// TwinCAT 3 PLC project PRINCIPAL
// Title: Programa Base 01
// Company: Escarre Automatizacion y Servecios sl
// ProjectVersion: 00_00
// ProgramVersion: 3.1.4023.0
// libraries:
//   EAS PLC, * (ESCARRE AUTOMATIZACION Y SERVICIOS sl)
//   EAS SCADA, * (ESCARRE AUTOMATIZACION Y SERVICIOS sl)
//   Tc2_Standard, * (Beckhoff Automation GmbH)
//   Tc2_SUPS, * (Beckhoff Automation GmbH)
//   Tc2_System, * (Beckhoff Automation GmbH)
//   Tc2_Utilities, * (Beckhoff Automation GmbH)
//   Tc3_Module, * (Beckhoff Automation GmbH)
//   Util, * (System)
// project tree:
//   DUTs/20_HARD/Beckhoff/ Island_Beck.TcDUT (not stored)
//   DUTs/20_HARD/ Hard.TcDUT
//   DUTs/MACHINE/DUT Elements/ dutAIn.TcDUT (not stored), dutAOut.TcDUT (not stored), dutPul.TcDUT, dutPump.TcDUT (not stored), dutValve.TcDUT (not stored)
//   DUTs/MACHINE/DUT System/ _00_GENERAL.TcDUT (not stored), _01_SEG.TcDUT (not stored), _02_TEMP.TcDUT, _03_PRESS.TcDUT (not stored), _04_FILL.TcDUT (not stored), _05_DRAIN.TcDUT, _06_LEVEL.TcDUT, _07_OVERFLOW.TcDUT, _08_CIRC.TcDUT (not stored), _09_CPUMP.TcDUT, _10_TK1.TcDUT, _11_TK2.TcDUT (not stored), _12_INTRO.TcDUT (not stored), _13_T_PREP.TcDUT (not stored), _14_CONSUM.TcDUT, _15_WINCH.TcDUT (not stored), _16_WINCH_X.TcDUT (not stored)
//   DUTs/MACHINE/ Machine.TcDUT
//   DUTs/10_PE/ ATL.TcDUT (not stored)
//   DUTs/10_PE/ELEMENTS/ PE.TcDUT (not stored), PE_COM.TcDUT
//   GVLs/ contants.TcGVL, Gloval_Variables.TcGVL (not stored), Mc.TcGVL (not stored), _Hard.TcGVL, _PE.TcGVL (not stored)
//   / PlcTask.TcTTO
//   POUs/00_Tasks/ ProgramaPrincipal.TcPOU
//   POUs/10_PE/ pComPE.TcPOU (not stored), pPE.TcPOU
//   POUs/20_Hardware/ pHard.TcPOU
//   POUs/30_PLC/30_1 UPS/ UPS.TcPOU
//   POUs/30_PLC/30_2 IO/ pIO.TcPOU
//   POUs/30_PLC/30_3_Config/ConfigSystem/ _00_Config_PE.TcPOU, _14_Config_Consum.TcPOU, _09_Config_CPump.TcPOU (not stored), _05_Config_Drain.TcPOU, _04_Config_Fill.TcPOU (not stored), _06_Config_LEVEL.TcPOU, _07_Config_Overflow.TcPOU (not stored), _03_Config_PRESS.TcPOU, _01_Config_SEG.TcPOU, _02_Config_TEMP.TcPOU (not stored), _10_Config_TK1.TcPOU (not stored), _11_Config_TK2.TcPOU (not stored), _15_Config_Winch.TcPOU, _00_Config_General.TcPOU (not stored)
//   POUs/30_PLC/30_3_Config/ pConfig.TcPOU
//   POUs/30_PLC/30_5_Funcions/Funcions/ F_AVISO.TcPOU, F_CARGA.TcPOU, F_CONTROL_PH.TcPOU, F_DESCARGA.TcPOU, F_DESPRESURIZA.TcPOU, F_DUCHAS.TcPOU (not stored), F_ESPERA.TcPOU (not stored), F_FIN_CICLO.TcPOU, F_FIN_DUCHAS.TcPOU (not stored), F_INTRO_TK2.TcPOU, F_ISOTERMA.TcPOU (not stored), F_LAVADO_CONT.TcPOU (not stored), F_LLENADO.TcPOU (not stored), F_LLENADO_TK2.TcPOU, F_MUESTRA.TcPOU, F_PREP_TK2.TcPOU, F_PRESURIZAR.TcPOU, F_RECIRCULA_TK2.TcPOU (not stored), F_TERMOREG.TcPOU (not stored), F_VACIADO.TcPOU (not stored), F_VACIADO_TK2.TcPOU, F_VELOCIDADES.TcPOU, _00_CIRC_PUMP.TcPOU (not stored), _00_CONSUMS.TcPOU (not stored), _00_GENERALES.TcPOU, _00_GESTION_PUL.TcPOU, _00_PID.TcPOU (not stored), _00_VENT.TcPOU
//   POUs/30_PLC/30_5_Funcions/ pFuctions.TcPOU
//   POUs/30_PLC/30_7 ActvOutputs/Modules/ Z_CIRC.TcPOU, z_CONTROL.TcPOU (not stored), Z_CP.TcPOU (not stored), z_DRAIN.TcPOU, z_FILL.TcPOU (not stored), Z_INTRO.TcPOU (not stored), z_LEVEL.TcPOU, z_OVERFLOW.TcPOU (not stored), z_PRESS.TcPOU, z_TEMP.TcPOU, z_TK1.TcPOU, z_TK2.TcPOU
//   POUs/30_PLC/30_7 ActvOutputs/ pActvOutputs.TcPOU
//   POUs/30_PLC/ ProgramPLC.TcPOU (not stored)
//   POUs/40_Function_Blocks/40_1_Llibreries_FB/ Canvi_Escala.TcPOU (not stored), Polsador.TcPOU, PULS_1S.TcPOU (not stored), TMP_P.TcPOU (not stored)
//   POUs/40_Function_Blocks/FB/Consums/ CONSUMP_00.TcPOU (not stored), KG_vapor_00.TcPOU (not stored), Kwh_00.TcPOU (not stored), Lit_H2O_00.TcPOU (not stored), Tabla_00.TcPOU (not stored)
//   POUs/40_Function_Blocks/FB/FB Duts/ fAI.TcPOU (not stored), fAO.TcPOU (not stored), fCaudal.TcPOU (not stored), fCnt.TcPOU (not stored), fTemp.TcPOU, fValve.TcPOU
//   POUs/40_Function_Blocks/FB/FB%27s_Utils/ fBCntLiters.TcPOU (not stored), fBHorn.TcPOU (not stored), fBPulse1s.TcPOU (not stored), fBUp_Down.TcPOU (not stored), fBWash_TK.TcPOU (not stored), fB_Intro_TK.TcPOU (not stored), fBPumpC.TcPOU (not stored), fBPumpSpeed.TcPOU (not stored), fBTermo.TcPOU (not stored)
//   Project Information/ F_GetCompany.TcPOU, F_GetTitle.TcPOU, F_GetVersion.TcPOU
// real-time tasks:
//   TASK PlcTask: cycle T#10ms, priority 20, ADS port 350
//   TASK PlcTask_1: cycle T#1ms, priority ?, ADS port 351
// I/O:
//   DEVICE Device 1 (EtherCAT), AmsNetId 5.110.215.44.2.1
//     Term 3 (EK1200) [EK1200-5000 EtherCAT Power supply (2A E-Bus)]
//       Term 1 (EL1512) [EL1512 2Ch. +/- Counter 24V, 1kHz]
//       Term 3 (EL1809) [EL1809 16Ch. Dig. Input 24V, 3ms]
//       Term 4 (EL1809) [EL1809 16Ch. Dig. Input 24V, 3ms]
//       Term 5 (EL1809) [EL1809 16Ch. Dig. Input 24V, 3ms]
//       Term 6 (EL2809) [EL2809 16Ch. Dig. Output 24V, 0.5A]
//       Term 7 (EL2809) [EL2809 16Ch. Dig. Output 24V, 0.5A]
//       Term 8 (EL2809) [EL2809 16Ch. Dig. Output 24V, 0.5A]
//       Term 9 (EL3202) [EL3202 2Ch. Ana. Input PT100 (RTD)]
//       Term 10 (EL3054) [EL3054 4Ch. Ana. Input 4-20mA]
//       Term 11 (EL4004) [EL4004 4Ch. Ana. Output 0-10V, 12bit]
//       Term 12 (EL9011) [EL9011 End Terminal]
//   DEVICE Device 4 (NOV-DP-RAM)
// variable links:
//   PRINCIPAL/PRINCIPAL Instance <-> Device 1 (EtherCAT)/Term 3 (EK1200)/Term 1 (EL1512)
//     PlcTask Inputs/pHard.CNT_Device[1] <-> CNT Inputs Channel 1/Counter value
//     PlcTask Inputs/pHard.CNT_Device[2] <-> CNT Inputs Channel 2/Counter value
//   PRINCIPAL/PRINCIPAL Instance <-> Device 1 (EtherCAT)/Term 3 (EK1200)/Term 10 (EL3054)
//     PlcTask Inputs/pHard.AI_Device[{3..6}] <-> AI Standard Channel {1..4}/Value  (4 links)
//   PRINCIPAL/PRINCIPAL Instance <-> Device 1 (EtherCAT)/Term 3 (EK1200)/Term 11 (EL4004)
//     PlcTask Outputs/pHard.AO_Device[{1..4}] <-> AO Outputs Channel {1..4}/Analog output  (4 links)
//   PRINCIPAL/PRINCIPAL Instance <-> Device 1 (EtherCAT)/Term 3 (EK1200)/Term 3 (EL1809)
//     PlcTask Inputs/pHard.DI_Device[{1..16}] <-> Channel {1..16}/Input  (16 links)
//   PRINCIPAL/PRINCIPAL Instance <-> Device 1 (EtherCAT)/Term 3 (EK1200)/Term 4 (EL1809)
//     PlcTask Inputs/pHard.DI_Device[{17..32}] <-> Channel {1..16}/Input  (16 links)
//   PRINCIPAL/PRINCIPAL Instance <-> Device 1 (EtherCAT)/Term 3 (EK1200)/Term 5 (EL1809)
//     PlcTask Inputs/pHard.DI_Device[{33..48}] <-> Channel {1..16}/Input  (16 links)
//   PRINCIPAL/PRINCIPAL Instance <-> Device 1 (EtherCAT)/Term 3 (EK1200)/Term 6 (EL2809)
//     PlcTask Outputs/pHard.DO_Device[{1..16}] <-> Channel {1..16}/Output  (16 links)
//   PRINCIPAL/PRINCIPAL Instance <-> Device 1 (EtherCAT)/Term 3 (EK1200)/Term 7 (EL2809)
//     PlcTask Outputs/pHard.DO_Device[{17..32}] <-> Channel {1..16}/Output  (16 links)
//   PRINCIPAL/PRINCIPAL Instance <-> Device 1 (EtherCAT)/Term 3 (EK1200)/Term 8 (EL2809)
//     PlcTask Outputs/pHard.DO_Device[{33..48}] <-> Channel {1..16}/Output  (16 links)
//   PRINCIPAL/PRINCIPAL Instance <-> Device 1 (EtherCAT)/Term 3 (EK1200)/Term 9 (EL3202)
//     PlcTask Inputs/pHard.AI_Device[1] <-> RTD Inputs Channel 1/Value
//     PlcTask Inputs/pHard.AI_Device[2] <-> RTD Inputs Channel 2/Value

CONFIGURATION PRINCIPAL
    RESOURCE PLC ON TwinCAT3
        TASK PlcTask(INTERVAL := T#10ms, PRIORITY := 20);
        PROGRAM ProgramaPrincipal WITH PlcTask : ProgramaPrincipal;
    END_RESOURCE
END_CONFIGURATION

// ---- DUTs/20_HARD/Hard.TcDUT
TYPE Hard :
STRUCT
	
Beck:ARRAY[1..Max_island_beck] OF Island_beck;

END_STRUCT
END_TYPE

// ---- DUTs/MACHINE/DUT Elements/dutPul.TcDUT
TYPE dutPul :
STRUCT
	xPul:BOOL;		// IN Pulsador
	xPil:BOOL;		// OUT Piloto

END_STRUCT
END_TYPE

// ---- DUTs/MACHINE/DUT System/_02_TEMP.TcDUT
TYPE _02_TEMP :
STRUCT
	///+++++++++++++++++++++++++++++++++++++++
	///HARD
	///+++++++++++++++++++++++++++++++++++++++
	v060_Aper: dutAOut;
	v061_Steam: dutValve;
	v062_Cool: dutValve;
	v063_RetCon: dutValve;
	v064_RecW: dutValve;
	s065_Reg: ftemp;
	s066_Mc: ftemp;
	s067_RetCon: ftemp;
	v068_Purge: dutValve;
	v069_AperCool: dutAout;
	/// Temperatura Maquina 
	rMacTemperature: REAL;
	///Temperatura  Impuesta
	rTempImp: REAL;
	///Señal para abrir retorno de condensados
	xRetCond: BOOL;
	/// PT100 Failure 
	xPT100Failure: BOOL;
	xMaxDifTemp: BOOL;
	///Gradiente por defecto
	iPFDefauldGrad: INT := 0;
	///Tiempo de bomba en m,archa para iniciar termorreg
	iPFTimeOfPumpToRun: INT := 60;
	///Grados para integracion
	iPFGradIntegra: INT := 2;
	///Grados para forzar calentamiento
	iPFGradForzCal: INT := 4;
	///Tiempo de seguridad para conmutacion vapor-frio
	iPFTmpComutac: INT := 30;
	///Grados para conmutacion en Mantenimiento
	iPFGradComutac: INT := 5;
	///PID_ Banda proporcional
	iPFPID_P: INT;
	///PID_ I= Parte integral
	iPFPID_I: INT;
	///PID_ D= Parte Derivada
	iPFPID_D: INT;
	///Temprearatura por debajo no se calienta
	iPFTempMinCool: INT := 45;
	
END_STRUCT
END_TYPE

// ---- DUTs/MACHINE/DUT System/_05_DRAIN.TcDUT
TYPE _05_DRAIN :
STRUCT
	///+++++++++++++++++++++++++++++++++++++++
	///HARD
	///+++++++++++++++++++++++++++++++++++++++
	v015_Grv: dutValve;
	v016_Grv2: dutValve;
	v017_Pump: dutValve;
	s018_LvlHT: dutPul;
	s019_TempHT: dutAIn;
	v020_HT: dutValve;
	v021_WaterHT: dutValve;
	///+++++++++++++++++++++++++++++++++++++++
	///READINGS
	///+++++++++++++++++++++++++++++++++++++++
	iTempHT: INT;
	xLvlHT: BOOL;
	///+++++++++++++++++++++++++++++++++++++++
	///PF - CONFIG
	///+++++++++++++++++++++++++++++++++++++++
	iPFMaxTimeDrain: INT;
	iPFTimeDrenado: INT;
END_STRUCT
END_TYPE

// ---- DUTs/MACHINE/DUT System/_06_LEVEL.TcDUT
TYPE _06_LEVEL :
STRUCT
	///+++++++++++++++++++++++++++++++++++++++
	///HARD
	///+++++++++++++++++++++++++++++++++++++++
	s031_Min: dutPul;
	s032_Perc: dutAIn;
	s033_max: dutPul;
	s034_L3: dutPul;
	s035_L2: dutPul;
	s036_L1: dutPul;
	v038_FillTb: dutValve;
	v039_DrainTb: dutValve;
	///Nivel de la maquina 0..100%
	rLevel: REAL;
	///Nivel 1 de la maquina
	xLvl_1: BOOL;
	///Nivel 2 de la maquina
	xLvl_2: BOOL;
	///Nivel 3 de la maquina
	xLvl_3: BOOL;
	///Nivel minimo de la maquina
	xLvl_min: BOOL;
	///Nivel maximo de la maquina
	xLvl_max: BOOL;
	///Nivel Alto de Recirculación
	xLvl_Wh: BOOL;
	///Nivel Bajoo de Recirculación
	xLvl_Wl: BOOL;
	///Fallo niveles
	xFailLvl: BOOL;
	///+++++++++++++++++++++++++++++++++++++++
	///PF - CONFIG
	///+++++++++++++++++++++++++++++++++++++++
	///Parametros configuracion Nivel analogico de Maquina
	iPFAna_min: INT := 0;
	iPFAna_max: INT := 100;
	///Porcentaje del nivel para bLvl_1
	iPFLvl_1: INT := 20;
	///Porcentaje del nivel para bLvl_2
	iPFLvl_2: INT := 50;
	///Porcentaje del nivel para bLvl_3
	iPFLvl_3: INT := 70;
	///Porcentaje del nivel para bLvl_min
	iPFLvl_min: INT := 0;
	///Porcentaje del nivel para bLvl_max
	iPFLvl_max: INT := 100;
	///Porcentaje del nivel alto de recirculación
	iPFLvl_Wh: INT := 60;
	///Porcentaje del nivel bajo de recirculación
	iPFLvl_Wl: INT := 20;
END_STRUCT
END_TYPE

// ---- DUTs/MACHINE/DUT System/_07_OVERFLOW.TcDUT
TYPE _07_OVERFLOW :
STRUCT
	///+++++++++++++++++++++++++++++++++++++++
	///HARD
	///+++++++++++++++++++++++++++++++++++++++
	v025_Valv: dutValve;
	v026_intrHT: dutValve;
	v027_VentHt: dutValve;
	v028_DrainHT: dutValve;
	v004_WaterInlet: dutValve;
	///Litros de la barcada
	rLit_Batch: REAL;
	///Litros Actuales
	rLit_Actual: REAL;
	///+++++++++++++++++++++++++++++++++++++++
	///CONFIG
	///+++++++++++++++++++++++++++++++++++++++
	iPFTimeFillAuxT: INT := 5;
	iPFTimeCloseAuzT: INT := 5;
	iPFTimeDepAuxT: INT := 5;
	iPFTimeDrainAuxT: INT := 5;
	iPFTimeCloseDrainAuxT: INT := 5;
END_STRUCT
END_TYPE

// ---- DUTs/MACHINE/DUT System/_09_CPUMP.TcDUT
TYPE _09_CPUMP :
STRUCT
	///+++++++++++++++++++++++++++++++++++++++
	///HARD
	///+++++++++++++++++++++++++++++++++++++++
	b450_CircPump: dutPump;
	p451_P_Run: dutPul;
	p452_P_Stop: dutPul;
	p453_P_AutoMan: dutPul;
	p454_P_UpVel: dutPul;
	p455_P_DownVel: dutPul;
	s456_Pote: dutAIn;
	p457_SelRun: dutPul;
	///+++++++++++++++++++++++++++++++++++++++
	///READINGS
	///+++++++++++++++++++++++++++++++++++++++
	rSP_Auto: REAL;
	rSP_Man: REAL;
	rSpeedUF: REAL;
	///+++++++++++++++++++++++++++++++++++++++
	///CONFIG
	///+++++++++++++++++++++++++++++++++++++++
	///++++PF+++
	iPF_AnaMax_UF: INT;
	iPF_AnaMin_UF: INT;
	iPF_AnaMax_perc: INT;
	iPF_AnaMin_perc: INT;
	iPF_SpeedMax_UF: INT;
	iPF_SpeedMin_UF: INT;
END_STRUCT
END_TYPE

// ---- DUTs/MACHINE/DUT System/_10_TK1.TcDUT
TYPE _10_TK1 :
STRUCT
	///+++++++++++++++++++++++++++++++++++++++
	///HARD
	///+++++++++++++++++++++++++++++++++++++++
	v101_Fill: dutValve;
	v102_RetMc: dutValve;
	v103_IntercTK: dutValve;
	b104_Intro: dutPump;
	v105_Drain_Pump: dutValve;
	v106_Drain_grav: dutValve;
	v107_Warm: dutValve;
	p108_Stirrer: dutPump;
	v109_Mixer: dutValve;
	v110_IntecIntro: dutValve;
	v111_Fill_TP: dutValve;
	v112_IntroTK2: dutValve;
	s113_Level: dutAin;
	s114_Temp: dutAin;
	o115_Lev1: dutPul;
	o116_Lev2: dutPul;
	p150_OKprod: dutPul;
	p151_P_Fill: dutPul;
	p152_P_Drain: dutPul;
	P153_P_RetMc: dutPul;
	p154_P_IntroFast: dutPul;
	p155_P_Warm: dutPul;
	p156_P_IntroSlow: dutPul;
	p157_P_Stirrer: dutPul;
	p158_P_Mixer: dutPul;
	p159_P_AutoMan: dutPul;
	p160_P_TK1_TK2: dutPul;
	///+++++++++++++++++++++++++++++++++++++++
	///READINGS
	///+++++++++++++++++++++++++++++++++++++++
	xLvl_min: BOOL;
	xLvl_max: BOOL;
	rLvl: REAL;
	xLvlHighCirc: BOOL;
	xLvlLowCirc: BOOL;
	xLvl_1: BOOL;
	xLvl_2: BOOL;
	xLvl_3: BOOL;
	rQt: REAL;
	rQr: REAL;
	///+++++++++++++++++++++++++++++++++++++++
	///CONFIG
	///+++++++++++++++++++++++++++++++++++++++
	iPFLvlAnaMin: INT;
	iPFLvlAnaMax: INT;
	iPFLvlMin: INT;
	iPFLvlMax: INT;
	iPFDescSonda: INT;
	iPFDreno: INT;
	iPF1rLav: INT;
	iPF2nLav: INT;
	iPF3rLav: INT;
	iPFDifAlarma: INT;
	iPFRetarBomba: INT;
	iPFHighCirc: INT;
	iPFLowCirc: INT;
	/// Volum Tank (Liters)
	iPFVolumTK: INT;
	iPFLvl_1: INT;
	iPFLvl_2: INT;
	iPFLvl_3: INT;
END_STRUCT
END_TYPE

// ---- DUTs/MACHINE/DUT System/_14_CONSUM.TcDUT
TYPE _14_CONSUM :
STRUCT
(*+++++++++++++++++++++++++++++++++++++++*)
(*HARD*)
(*+++++++++++++++++++++++++++++++++++++++*)
	s500_Amperimetre	:dutAin;


	
(*+++++++++++++++++++++++++++++++++++++++*)
(*READINGS*)
(*+++++++++++++++++++++++++++++++++++++++*)

	rLit_Batch		:REAL;		(*Litros de la barcada*)
	rKw_Batch		:REAL; 		(*Kw de la Barcada*)
	rKgStm_Batch	:REAL;		(*Kg de Vapor de la barcada*)
	rAmp			:REAL;		//Corriente de entrada


(*+++++++++++++++++++++++++++++++++++++++*)
(*CONFIG*)
(*+++++++++++++++++++++++++++++++++++++++*)




	
END_STRUCT
END_TYPE

// ---- DUTs/MACHINE/Machine.TcDUT
TYPE Machine :
STRUCT
	///Sistema de Batch
	_00_GENERAL: _00_GENERAL;
	///SEGURIDAD
	_01_SEG: _01_SEG;
	///Sistema de calentamiento
	_02_TEMP: _02_TEMP;
	///Sistema de PRESURITZACIÓ
	_03_PRESS: _03_PRESS;
	///Sistema de llenado
	_04_FILL: _04_FILL;
	///Sistema de Vaciado
	_05_DRAIN: _05_DRAIN;
	///Sistema de Niveles de la maquina
	_06_LEVEL: _06_LEVEL;
	///Sistema de Rebosadero
	_07_OVERFLOW: _07_OVERFLOW;
	///Valvulas de la circulacion
	_08_CIRC: _08_CIRC;
	///Bomba de circulacion
	_09_CPUMP: _09_CPUMP;
	///Tanque 1
	_10_TK1: _10_TK1;
	///Tanque 2
	_11_TK2: _11_TK2;
	///Sistema de Intorduccion
	_12_INTRO: _12_INTRO;
	///Tanque Preparacion
	_13_TPrep: _13_T_PREP;
	///Sistema de Consumos
	_14_CONSUM: _14_CONSUM;
	///Troniquetes
	_15_WINCH: _15_WINCH;
	

	
	
END_STRUCT
END_TYPE

// ---- DUTs/10_PE/ELEMENTS/PE_COM.TcDUT
TYPE PE_COM :
STRUCT
	
(* -------------------------------------------------------------------- *)
(* InfoBarcada *)
	sBatch:STRING[10];			
	diNum_Task:DWORD;
	sCdRecipe:STRING[24];
	sDesc_Recipe:STRING[50];
	sCdCycle:STRING[10];
	sDesc_Cycle:STRING[50];

(* -------------------------------------------------------------------- *)
(* Ordenes PE *)
	xToAutomatic	:BOOL;
	xToManual		:BOOL;
	xToStep			:BOOL;
	xRunCycle		:BOOL;
	xModifiedCycle	:BOOL;
	xStopAlarm		:BOOL;
	xContProg		:BOOL;		 	(*Bit Para continuar programa*)
	xStartTopping	:BOOL;			(*Bit indicacion al iniciar una añadida*)
	xEndTopping		:BOOL;			(*Bit indicacion al finalizar una añadida*)
	xResetStep		:BOOL;			(*Bit indicacion para resetar los tiempos de la funcion al realizar un salto*)
	xReset			:BOOL;
	xResetFunc		:BOOL;
	wNewStep		:WORD;			(*word Per fer un canvi de Pas*)

	
	
(* -------------------------------------------------------------------- *)
(* Dosificacio *)
	
	axDemandDos		: ARRAY [1..max_tanks] OF BOOL;	; 		(* Pedir Dosificacion*)
	aiNumDos		: ARRAY [1..max_tanks] OF WORD;			(* Numero Dosificacion *)
	axOkDemand		: ARRAY [1..max_tanks] OF BOOL;			(* OK Peticion Dosificacion*)	
	axOkDosage		: ARRAY [1..max_tanks] OF BOOL;			(* OK  Dosificacion*)	
	aiTypeDos		: ARRAY [1..max_tanks] OF WORD;	 	  	(* Tipo Dosificacion 1=Man 2=Auto 3=Mixta*)
	axProdMan		: ARRAY [1..max_tanks] OF BOOL;			(* Dosificacion con Producto  Manual **)	
	axErrorDos		: ARRAY [1..max_tanks] OF BOOL;			(* Error Dosificación  **)	
	aiVolumDos		: ARRAY [1..max_tanks] OF DWORD;		(* Volumen dosificat*)
	axTankFree		: ARRAY [1..max_tanks] OF BOOL;			(* Tanque libre *)
	aiPriority		: ARRAY [1..max_tanks] OF WORD;			(* Prioridad*)
	axOnlyDissol	: ARRAY [1..max_tanks] OF BOOL;			(* Solo Disolver*)





	
(* -------------------------------------------------------------------- *)
	
//	No utilizadas:
//	ActivarParalelo:BOOL;
//	DesactivarParalelo:BOOL;



END_STRUCT
END_TYPE

// ---- GVLs/contants.TcGVL
VAR_GLOBAL CONSTANT

(*=======================================	*)
(*			Carregar Constants						*)
(*=======================================	*)
	max_Funcions:WORD:=64;
	max_ParamFunc:WORD:=9;
	max_FinFunc:WORD:=5;
	max_PasCicle:WORD:=256;
	Max_Compatibles:WORD:=32;
	Max_Func_Pas:WORD:=12;
	Max_Alarmes:WORD:=128;
	Max_ParamFixes:WORD:=150;
	Max_DBFiFuncio: WORD:=320 ;				(* Es calcula com    (Max_Funcions*Max_FinFunc)   *)
	Max_ElementsCicle: WORD:=2816 ;		(* Es calcula com    (Max_PasCicle*(Max_ParamFunc+2))  *)
	Max_DBIncompatibles: WORD:=64;			(* Es calcula com    (Max_Compatibles*2)  *)
	Max_Inputs: WORD:=128;
	Max_Outputs: WORD:=128;
	Max_Analog: WORD:=32;
	Num_Prod_Dos:WORD:=10;         					(* Numero maximo de productos en una dosificación*)
	Max_Prod_Dos:WORD:=128;							(* Productos en una dosificadora*)
	Max_Valv_Dos:WORD:=128;							(* Valvulas en una do*)
	Max_Tanks:WORD:=4;
	
	
(*=======================================	*)
(*			Hardware Beckhoff				*)
(*=======================================	*)
	Max_island_beck	:WORD:=5;
	Max_DI_Beck		:WORD:=256;
	Max_DO_Beck		:WORD:=256;
	Max_AI_Beck		:WORD:=32;
	Max_AO_Beck		:WORD:=32;
	Max_CNT_Beck	:WORD:=16;
	
	     
	
END_VAR

// ---- GVLs/_Hard.TcGVL

VAR_GLOBAL 
HARD:Hard;
	

END_VAR

// ---- POUs/00_Tasks/ProgramaPrincipal.TcPOU
PROGRAM ProgramaPrincipal
VAR
	azzz: WORD;
	pols:R_TRIG;
	azzz_ant: WORD;
	cont_scan_2s: WORD;
END_VAR

(*=============================================================*)
(*									++++++++									*)
(*								Programa Principal  							*)
(*									++++++++									*)
(*=============================================================*)

(* Control de run *)
azzz:=azzz+1;
IF azzz>999
	THEN
		azzz:=0;
END_IF


(* -------------------------------------------------------------------------------------------------------------*)
(* 			Pe4																		*)
(* -------------------------------------------------------------------------------------------------------------*)

pComPe();
 


(* -------------------------------------------------------------------------------------------------------------*)
(* 			Gestió del Cicle														*)
(* -------------------------------------------------------------------------------------------------------------*)

pPE();


(* -------------------------------------------------------------------------------------------------------------*)
(* 			Configuracion Hard																		*)
(* -------------------------------------------------------------------------------------------------------------*)


pHard();

(* -------------------------------------------------------------------------------------------------------------*)
(* 			PLC																		*)
(* -------------------------------------------------------------------------------------------------------------*)


ProgramPLC();

END_PROGRAM

// ---- POUs/10_PE/pPE.TcPOU
PROGRAM pPE
VAR PERSISTENT
	Anar1:Salt;
	Anar2:Salt;
	Anar3:Salt;
	Anar4:SaltDePasEnUnCicle;
	Anar5:SaltDePasEnUnCicle;
	Parar:PararTotesLesFuncions;
	PararInici:PararTotesLesFuncions;
	ComprobarSalt:ComprobarFuncionsPas;
	SaltarProximPas:BOOL;
	EsperaSalt:TON;
	AcualitzaDB: CarregarFuncionsActivesAlDB;
	AcualitzaDB2: CarregarFuncionsActivesAlDB;
	PunterCicle0: WORD;
	ferSalt: BOOL;
	FerSaltParalel: BOOL;    (*ordre de salt*)
	EsperaSaltar: TON;
	SaltarPar: BOOL;
	PararTot:PararTotesLesFuncions;
	

(*=========================================================*)	
(*========  GESTIÓ MANUAL  ================================*)	

	Punt_Func: WORD;
	T_Func_Act:T_Funcio;				(* Funcio que indica el punterCicle *)
	FiFuncio:Parar_Func_FiFuncio;
	Incompatibles: Parar_Func_Incomp;
	a: WORD;
	AcualitzaDB3: CarregarFuncionsActivesAlDB;
	

(*=========================================================*)	
	fbFUNBCK: FunBck_v01;
	xFunBck: BOOL;
	tFunBck: Ton;
	tCicloOn: ton;
	rsBatch: Rs;
	
END_VAR
VAR
	run:BOOL;
	inici: Ton;
	fb_UPS_CX8190: FB_S_UPS_CX81xx;
	xCargadas: BOOL;
	xUltimas: BOOL;
	xBackup: BOOL;
	END_VAR

(*==============================================================*)
(*		GESTION REMANENTES PARA CPU CX8190  					*)
(*==============================================================*)
(*
fb_UPS_CX8190(
	sNetID:= , 
	iPLCPort:=851 , 
	tTimeout:= , 
	eUpsMode:= , 
	ePersistentMode:= , 
	tRecoverTime:= , 
	bPowerFailDetect=> , 
	eState=> );

IF _AppInfo.BootDataLoaded THEN
	xCargadas:=TRUE;
	ELSE
		xCargadas:=FALSE;
END_IF

IF _AppInfo.OldBootData THEN
	xUltimas:=FALSE;
	xBackup:=TRUE;
	ELSIF _AppInfo.BootDataLoaded THEN
		xUltimas:=TRUE; 
		xBackup:=FALSE;
END_IF


*)


(*==============================================================*)
(*		GESTION PE												*)
(*==============================================================*)
(*,,,,,,,,,,,,,,,,,,,,,,,,,,,,,,,,,,,,,,,,,,,,,Pasar a manual al reiniciar  ,,,,,,,,,,,,,,,,,,,,,,,,,,,,,,,,,,,,,,,,,,,,,,,	*)
inici(IN:= run, PT:=T#5S , Q=> , ET=> );


IF NOT inici.Q THEN
ATL.PE_COM.xToManual:=TRUE;
ATL.PE.wAutoMan:=1;
ATL.PE_COM.xResetFunc:=TRUE;
PararInici(Estat_F:=est_func );
run:=TRUE;
END_IF



(*,,,,,,,,,,,,,,,,,,,,,,,,,,,,,,,,,,,,,,,,,,,,, Orde de Ejecutar Cicle    ,,,,,,,,,,,,,,,,,,,,,,,,,,,,,,,,,,,,,,,,,,,,,,,,,,,,	*)

IF ATL.PE_COM.xRunCycle
	THEN
		Cicle0:=CicleRebut;
		ATL.PE.wStep :=0;
		ATL.PE.wAutoMan:=2;
		Anar2(
			PasInicial:= 0 ,
			 PasFinal:= ATL.PE.wStep );
		ATL.PE_COM.xRunCycle:= FALSE;
END_IF

(*,,,,,,,,,,,,,,,,,,,,,,,,,,,,,,,,,,,,,,,,,,,,,Orde de Cicle Modificat ,,,,,,,,,,,,,,,,,,,,,,,,,,,,,,,,,,,,,,,,,,,,,,,,	*)
IF ATL.PE_COM.xModifiedCycle
	THEN
		Cicle0:=CicleRebut;
		ATL.PE_COM.xModifiedCycle:=FALSE;
END_IF

(*,,,,,,,,,,,,,,,,,,,,,,,,,,,,,,,,,,,,,,,,,,,,,Orde de Reset ,,,,,,,,,,,,,,,,,,,,,,,,,,,,,,,,,,,,,,,,,,,,,,,,,,,,,,,,,,,,,,,,	*)
IF ATL.PE_COM.xReset
	THEN
		PararTot(Estat_F:=Est_F_PE4 );
		ATL.PE.wStep :=0;
		ATL.PE_COM.xToManual:=TRUE;
		ATL.PE_COM.xReset:=FALSE;
END_IF
(*,,,,,,,,,,,,,,,,,,,,,,,,,,,,,,,,,,,,,,,,,,,,,Orde de Reset ,,,,,,,,,,,,,,,,,,,,,,,,,,,,,,,,,,,,,,,,,,,,,,,,,,,,,,,,,,,,,,,,	*)
IF ATL.PE_COM.xResetFunc
	THEN
		PararTot(Estat_F:=Est_F_PE4 );
		ATL.PE_COM.xResetFunc :=FALSE;
END_IF


(*=============================================================*)
(*=============================================================*)

(*Control si el sistema treballa en MANUAL / AUTOMATIC *)

(*,,,,,,,,,,,,,,,,,,,,,,,,,,,,,,,,,,,,,,,, Canvis d'estat AUTO/MAN ,,,,,,,,,,,,,,,,,,,,,,,,,,,,,,,,,,,,,,,,,,,,,,,,,	*)
(*  Automàtic   *)
IF ((ATL.PE.xPulAuto)(*OR Com_PE.RetardArranc*) OR (ATL.PE_COM.xToAutomatic) OR (ATL.PE.wAutoMan>2))AND(cicle0[1].Pas<>0)
	THEN
		(* Pasar de Manual a Automatic*)
		IF ATL.PE.wAutoMan<=1
			THEN
				Parar(Estat_F:=Est_Func);
				IF ATL.PE.wStep=0
					THEN
						ATL.PE.wStep:=1;
				END_IF
				Anar3(
					PasInicial:= 0 ,
		 			PasFinal:= ATL.PE.wStep );
		END_IF
		ATL.PE.wAutoMan:=2;
		AcualitzaDB
			(EstatFuncions:= Est_Func  ,
			FuncionsActives=>Func_Actives );
END_IF;
		ATL.PE_COM.xToAutomatic:=FALSE;

(*  Manual   *)
IF (ATL.PE.xPulMan) OR (ATL.PE_COM.xToManual) OR (ATL.PE.wAutoMan<1)
	THEN
		(* Pasar d'automatic a manual *)
		IF ATL.PE.wAutoMan>=2
			THEN
				Parar(Estat_F:=Est_Func);
		END_IF
		ATL.PE.wAutoMan:=1;
		ATL.PE_COM.xToManual:=FALSE;
END_IF;


(*=============================================================*)
(* + + + + + + + +  +  + + + + + + + + + + + + + + + + + + + + + + + + + + + + + + + + + *)

(*,,,,,,,,,,,,,,,,,,,,,,,,,,,,,,,,,,,,,,,,,, Gestio Manual,,,,,,,,,,,,,,,,,,,,,,,,,,,,,,,,,,,,,,,,,,,,,,,,,,,,,,,,,,,,,,,,,,,,,	*)

IF ATL.PE.wAutoMan=1
	THEN
(*_____________________________________________________________________________________________________________*)
		Punt_Func:=1;
		REPEAT
			IF (Est_Func[Punt_Func].Actv_Funcio)=(Est_F_PE4[Punt_Func].Actv_Funcio)
			THEN
				(*Igualar valors de les funcions*)
				Est_Func[Punt_Func]:=Est_F_PE4[Punt_Func];
				(*Aumentar el punter*)
				Punt_Func:=Punt_Func+1;
			ELSE
				T_Func_Act:=Config_Func[Punt_Func];
				IF Est_Func[Punt_Func].Actv_Funcio=TRUE
				THEN
					(* Parar la funcio al PLC per fi funcio manual al PE4  *)
					Est_Func[Punt_Func].Actv_Funcio:=FALSE;
				ELSE
					IF (Est_F_PE4[Punt_Func].Actv_Funcio=TRUE)AND(Est_F_PE4_Ant[Punt_Func].Actv_Funcio=TRUE)
					THEN
						(*Parar la funcio al PE4 per que s'ha acabat*)
							Est_F_Pe4[Punt_Func].Actv_Funcio:=FALSE;
					ELSE
						(*=====Activar la funció====*)
						(*Mirar si hi ha alguna funció incompatible amb la nova funció*)
						Incompatibles(
							Funcio:= T_Func_Act.Cd_funcio ,
							DB_Comp:= Func_Comp,
							Estat_F:=Est_Func );
		
						(*Mirar si la funcio nova ha d'acabar alguna funció per Fin Funcion*)
						FiFuncio(
							Tipus_Funcio:= T_Func_Act ,
							Estat_F:= Est_func);
						(*Activar la funció*)
						Est_Func[Punt_Func]:= Est_F_PE4[Punt_Func];
					END_IF
				END_IF
			END_IF
		UNTIL
		Punt_Func>Max_Funcions
		END_REPEAT
		AcualitzaDB3
			(EstatFuncions:= Est_Func  ,
			FuncionsActives=>Func_Actives );
		
		Est_F_PE4_Ant:=Est_F_PE4;
(*_____________________________________________________________________________________________________________*)
		SaltarProximPas:=FALSE;
END_IF


(*=============================================================*)
(* + + + + + + + +  +  + + + + + + + + + + + + + + + + + + + + + + + + + + + + + + + + + *)
(*,,,,,,,,,,,,,,,,,,,,,,,,,,,,,,,,,,,,, Gestio En Autiomatic,,,,,,,,,,,,,,,,,,,,,,,,,,,,,,,,,,,,,,,,,,,,,,,,,,,,,,,,,,,,,	*)


IF ATL.PE.wAutoMan=2
	THEN
		(*__________________Comprobar si cal pasar la seguent PAS_______________________________________________*)
		ComprobarSalt(
			Estat_F:= Est_Func,
			Tipus_F:=Config_Func ,
			FuncionsActives:= Func_Actives,
			AumentaPas=> SaltarProximPas );

		(*__________________Buscar Punter Cicle del pas inicial___________________________________________________*)

	PunterCicle0:=0;
		REPEAT
			PunterCicle0 := PunterCicle0+1;
		UNTIL
			(((Cicle0[PunterCicle0].Pas=ATL.PE.wStep)AND(Cicle0[PunterCicle0+1].Pas<>ATL.PE.wStep)) OR (PunterCicle0>=max_PasCicle))
		END_REPEAT

		(*__________________Fer Canvi de pas _______________________________________________________________*)
		IF SaltarProximPas AND NOT he_C_local
			THEN
				IF NOT(MaquinaEnParalel)
				THEN
				(* ·······················Maquina Single o Paralel desacoplada ··············································································································· *)
				Anar4(
					PasInicial:= ATL.PE.wStep,
		 			PasFinal:= (ATL.PE.wStep + 1) );
				ATL.PE.wStep:=ATL.PE.wStep + 1;
				SaltarProximPas:=FALSE;
				AcualitzaDB(
					EstatFuncions:= Est_Func  ,
					FuncionsActives=>Func_Actives );
				ELSE
				(* ·······················Maquina  En Paralel Acoplada ··························································································································· *)
				(*---------------------------------------------------------------------------------------------------------------------------------------------------------*)
				(*........................Indicar que la maquina local està preparada per pasar de pas..........................:........................................*)
				Preparat_C_local:=TRUE;
				(*........................Ordre de canvi ::::..........::::::::::.........::::::::::.........::::::::::.........::::::::::.........::::::::::.........::::::::::.........::::::::::.........:::::.*)
				(*........................Maquina Master: Actv ordre de canvi de pas.::::::::::.........::::::::::.........::::::::::.........::::::::::.........::::::::::.........:::::.*)
				(* 10/06/2011   preparat per diferents tipus de paralel   *)
				IF tipoparalelo<=2 THEN
					Ordre_C:= Master AND Preparat_C_local AND Preparat_C_S1;
				END_IF
				IF tipoparalelo=3 THEN
					Ordre_C:= Master AND Preparat_C_local AND Preparat_C_S1 AND Preparat_C_S2;
				END_IF
				IF tipoparalelo=4 THEN
					Ordre_C:= Master AND Preparat_C_local AND Preparat_C_S1 AND Preparat_C_S2 AND Preparat_C_S3;
				END_IF
				IF tipoparalelo>=5 THEN
					Ordre_C:= Master AND Preparat_C_local AND Preparat_C_S1 AND Preparat_C_S2 AND Preparat_C_S3 AND Preparat_C_S4;
				END_IF

				(*........................Activar el canvi procedent del master ..........::::::::::.........::::::::::.........::::::::::.........::::::::::.........::::::::::.........:::::.*)
				FerSaltParalel:=Ordre_C_Master AND NOT He_C_local;
				(*"""""""""""""Ordre de saltar,,,,,,,,,,,,,,,,,,,,,,,,,,,,,,,,,,,,,,,,,,,,,,,,,,,,,,,,,,,,,,,,,,,,,,,,,,,,,,,,,,,,,,,,,,,,,,,,,,,,,,,,,,,,,,,,,,,,,,,,,,,,,,,,,,,,,,,,,,,,,,,,,,,,,,,,,,,,,,*)
				IF  SaltarPar THEN
					Anar5(
						PasInicial:= ATL.PE.wStep,
		 				PasFinal:= (ATL.PE.wStep+1) );
					ATL.PE.wStep:=ATL.PE.wStep+1;
					SaltarProximPas:=FALSE;
					AcualitzaDB2(
						EstatFuncions:= Est_Func  ,
						FuncionsActives=>Func_Actives );
				(*........................Marca local  que ja s'ha fet el salt ::::..........::::::::::.........::::::::::.........::::::::::.........::::::::::.........::::::::::.........:::::.*)
					He_C_local:=TRUE;                            (* Marca de salt fet *)
				END_IF
			END_IF
		END_IF
		Est_F_PE4_Ant:=Est_F_PE4;
		Est_F_PE4:=Est_Func;
END_IF

(*Espera per asegurar que no es fa més de un salt de cop*)
EsperaSaltar(IN:= FerSaltParalel, PT:=t#1s , Q=>SaltarPar );

(*........................Maquina Master: Comprobar que tots han fet el canvi:::::::::.........::::::::::.........::::::::::.........::::::::::.........:::::.*)
(* 10/06/2011   preparat per diferents tipus de paralel   *)
IF tipoparalelo<=2 THEN
	Fi_C:= ( Master AND He_C_local AND He_C_S1 )OR( master AND Fi_C AND Preparat_C_S1);
END_IF
IF tipoparalelo=3 THEN
	Fi_C:= ( Master AND He_C_local AND He_C_S1 AND He_C_S2 )OR( master AND Fi_C AND (Preparat_C_S1 OR Preparat_C_S2));
END_IF
IF tipoparalelo=4 THEN
	Fi_C:= ( Master AND He_C_local AND He_C_S1 AND He_C_S2 AND He_C_S3 )OR( master AND Fi_C AND (Preparat_C_S1 OR Preparat_C_S2 OR Preparat_C_S3));
END_IF
IF tipoparalelo>=5 THEN
	Fi_C:= ( Master AND He_C_local AND He_C_S1 AND He_C_S2 AND He_C_S3 AND He_C_S4 )OR( master AND Fi_C AND (Preparat_C_S1 OR Preparat_C_S2 OR Preparat_C_S3 OR Preparat_C_S4));
END_IF



(*........................Fer Reset dels valors per fi de canvi de pas::::::::::::::::::::::::::.........::::::::::.........::::::::::.........::::::::::.........:::::.*)
IF Fi_C_Master OR ATL.PE.wAutoMan<=1 OR NOT(MaquinaEnParalel) THEN
	Preparat_C_local:=FALSE;
	Preparat_C_S1:=FALSE;
	Preparat_C_S2:=FALSE;
	Preparat_C_S3:=FALSE;
	Preparat_C_S4:=FALSE;
	He_C_local:=FALSE;
	He_C_S1:=FALSE;
	He_C_S2:=FALSE;
	He_C_S3:=FALSE;
	He_C_S4:=FALSE;
	Ordre_C:=FALSE;
	Ordre_C_Master:=FALSE;
	FerSaltParalel:=FALSE;
	SaltarPar:=FALSE;
END_IF

(* Reset valors paralel en cas de manual*)
IF ATL.PE.wAutoMan=1
	THEN
	FerSaltParalel:=FALSE;
END_IF

(*,,,,,,,,,,,,,,,,,,,,,,,,,,,,,,,,,,,,,,,,,,,,,Orde de Salt de pas ,,,,,,,,,,,,,,,,,,,,,,,,,,,,,,,,,,,,,,,,,,,,,,,,,,,,,,,,	*)
EsperaSalt(IN:= ATL.PE_COM.xToStep, PT:=T#2S , Q=>ferSalt , ET=> );
IF ferSalt 
	THEN
		Parar(Estat_F:= Est_Func );
		Anar1(
			PasInicial:= 0 ,
			PasFinal:= ATL.PE_COM.wNewStep );
		ATL.PE.wStep:=ATL.PE_COM.wNewStep;
		ATL.PE_COM.xResetStep:=TRUE;
		ATL.PE_COM.xToStep:= FALSE;
END_IF
AcualitzaDB(
	EstatFuncions:= Est_Func  ,
	FuncionsActives=>Func_Actives );


(*=====================================================================================================================================*)
(* INDICACIONS AUTO MAN*)

ATL.PE.xMan := ATL.PE.wAutoMan= 1  ;
ATL.PE.xAuto := ATL.PE.wAutoMan= 2  ;

(*=====================================================================================================================================*)
(*CALCULO DURACION PASO*)
fbFUNBCK(funcioBck=>xFunBck );
tFunBck(IN:=xFunBck , PT:=T#10D );
ATL.PE.wTStep := REAL_TO_WORD((TIME_TO_REAL(tFunBck.ET))/1000.0); (*expresado en segundos*)
(*=====================================================================================================================================*)
(*CALCULO DURACION BARCADA*)
rsBatch(SET:=ATL.PE.xStartBatch , RESET1:=ATL.PE.xEndBatch );
tCicloOn(IN:= rsBatch.Q1, PT:=T#10D );
ATL.PE.wTBatch:= REAL_TO_WORD((TIME_TO_REAL(tCicloOn.ET))/60000.0);(*expresado en minutos*)
(*=====================================================================================================================================*)

END_PROGRAM

// ---- POUs/20_Hardware/pHard.TcPOU
PROGRAM pHard
VAR
	DI_Device AT %I*: ARRAY[1..Max_DI_Beck] OF BOOL;
	DO_Device AT %Q*: ARRAY[1..Max_DO_Beck] OF BOOL;
	AI_Device AT %I*: ARRAY[1..Max_AI_Beck] OF INT;
	AO_Device AT %Q*: ARRAY[1..Max_AO_Beck] OF INT;
	CNT_Device AT %I*: ARRAY[1..Max_CNT_Beck] OF UDINT;
	Borrar:BOOL;
	
	iPunt: WORD;
END_VAR


(*==============================================================
1001= DI
1002= DO
1003= AI 0..10V
1004= AI 4..20mA
1005= AO 0..10V
1006= AO 4..20mA
1007= AI pt-100
1008= CNT

===================================================================*)

(*==============================================================
1001= DI
1002= DO
1003= AI 0..10V
1004= AI 4..20mA
1005= AO 0..10V
1006= AO 4..20mA
1007= AI pt-100
1008= CNT

===================================================================*)(*-------------------------------------------------------------------------*)
(*CArgar configuracion Beckhoff a la variable HArd*)
(*-------------------------------------------------------------------------*)
(*DI*)
iPunt:=1;
WHILE ipunt< Max_DI_Beck+1
	DO
	hard.Beck[1].DIN[iPunt]:=DI_Device[ipunt];
	iPunt:=iPunt+1;
END_WHILE
(*-------------------------------------------------------------------------*)
(*DO*)
iPunt:=1;
WHILE ipunt< Max_DO_Beck+1
	DO
	DO_Device[ipunt]:=hard.Beck[1].DOUT[iPunt];
	iPunt:=iPunt+1;
END_WHILE
(*-------------------------------------------------------------------------*)
(*AI*)
iPunt:=1;
WHILE ipunt< Max_AI_Beck+1
	DO
	hard.Beck[1].AIN[iPunt]:=AI_Device[ipunt];
	iPunt:=iPunt+1;
END_WHILE
(*-------------------------------------------------------------------------*)
(*AO*)
Borrar:=TRUE;
iPunt:=1;
WHILE ipunt< Max_AO_Beck+1
	DO
	AO_Device[ipunt]:=REAL_TO_INT(hard.Beck[1].AOUT[iPunt]);
	iPunt:=iPunt+1;
END_WHILE

(*-------------------------------------------------------------------------*)
(*CNT*)
iPunt:=1;
WHILE ipunt< Max_CNT_Beck+1
	DO
	hard.Beck[1].CNT[iPunt]:=CNT_Device[ipunt];
	iPunt:=iPunt+1;
END_WHILE
(*-------------------------------------------------------------------------*)

END_PROGRAM

// ---- POUs/30_PLC/30_1 UPS/UPS.TcPOU
PROGRAM UPS
VAR
	run:BOOL;
	
	fb_UPS_CX8190: FB_S_UPS_CX81xx;
	fb_UPS_CX9020: FB_S_UPS_CX9020_U900;
	xCargadas: BOOL;
	xUltimas: BOOL;
	xBackup: BOOL;
END_VAR

(*==============================================================*)
(*		GESTION REMANENTES PARA CPU CX8190 O CX9020 					*)
(*==============================================================*)
(*
fb_UPS_CX8190(
	sNetID:= , 
	iPLCPort:=851 , 
	tTimeout:= , 
	eUpsMode:= , 
	ePersistentMode:= , 
	tRecoverTime:= , 
	bPowerFailDetect=> , 
	eState=> );*)
	
	fb_UPS_CX9020(
	sNetID:= , 
	iPLCPort:=851 , 
	tTimeout:= , 
	eUpsMode:= , 
	ePersistentMode:= , 
	tRecoverTime:= , 
	bPowerFailDetect=> , 
	eState=> );

IF _AppInfo.BootDataLoaded THEN
	xCargadas:=TRUE;
	ELSE
		xCargadas:=FALSE;
END_IF

IF _AppInfo.OldBootData THEN
	xUltimas:=FALSE;
	xBackup:=TRUE;
	ELSIF _AppInfo.BootDataLoaded THEN
		xUltimas:=TRUE; 
		xBackup:=FALSE;
END_IF

END_PROGRAM

// ---- POUs/30_PLC/30_2 IO/pIO.TcPOU
PROGRAM pIO
VAR
	Cargar: INT;
	aaa: INT;
	MANUAL: INT;
	AA: REAL;
END_VAR


(*======================================================================*)
(*			COUNTER INPUTS												*)
(*======================================================================*)
MC._04_FILL.s010_Flowm.iCnt  			:= hard.Beck[1].CNT[1];
//MC.CONSUM.s500_Amperimetre.R	:= hard.Beck[1].CNT[2];
(*======================================================================*)
(*			DIGITAL INPUTS												*)
(*======================================================================*)
(*========= MODULO 2 ===================================================*)

Mc._00_GENERAL.p400_PMAn.xPul			:= hard.Beck[1].DIN[1];
Mc._00_GENERAL.p401_PAuto.xPul			:= hard.Beck[1].DIN[2];
Mc._00_GENERAL.p402_StopAlarm.xPul		:= hard.Beck[1].DIN[3];
Mc._00_GENERAL.p403_ContProg.xPul		:= hard.Beck[1].DIN[4];
Mc._00_GENERAL.p411_FailPump.xPul		:= hard.Beck[1].DIN[5];  				 
Mc._01_SEG.s420_MaxPresTemp.xPul		:= hard.Beck[1].DIN[6];
Mc._01_SEG.s421_BloqValv.xPul			:= hard.Beck[1].DIN[7];
Mc._06_LEVEL.s031_Min.xPul				:= hard.Beck[1].DIN[8];
Mc._01_SEG.s422_McClose.xPul			:= hard.Beck[1].DIN[9];
//Mc._00_GENERAL.p400_PMAn.xPul	 		:= hard.Beck[1].DIN[10];
mc._06_LEVEL.s036_L1.xPul				:= hard.Beck[1].DIN[11];
Mc._06_LEVEL.s035_L2.xPul				:= hard.Beck[1].DIN[12];
Mc._06_LEVEL.s034_L3.xPul				:= hard.Beck[1].DIN[13];
Mc._15_WINCH.W[1].s07_Tangle.xPul		:= hard.Beck[1].DIN[14];
Mc._15_WINCH.W[2].s07_Tangle.xPul		:= hard.Beck[1].DIN[15];					
//Mc._15_WINCH.W[1].p00_Winch.xInCons	:= hard.Beck[1].DIN[16];			  

(*========= MODULO 3 ===================================================*)

Mc._09_CPUMP.p451_P_Run.xPul		:= hard.Beck[1].DIN[17];	
Mc._09_CPUMP.p452_P_Stop.xPul			:= hard.Beck[1].DIN[18];
Mc._09_CPUMP.b450_CircPump.xInCons		:=true;//:= hard.Beck[1].DIN[19];
Mc._09_CPUMP.p453_P_AutoMan.xPul		:= hard.Beck[1].DIN[20];
Mc._09_CPUMP.p455_P_DownVel.xPul		:= hard.Beck[1].DIN[21]; 
Mc._09_CPUMP.p454_P_UpVel.xPul			:= hard.Beck[1].DIN[22];	
Mc._15_WINCH.W[1].p01_Run.xPul			:= hard.Beck[1].DIN[23];
Mc._15_WINCH.W[1].p02_Rev.xPul			:= hard.Beck[1].DIN[24];
Mc._15_WINCH.W[1].P03_AutoMan.xPul		:= hard.Beck[1].DIN[25];
Mc._15_WINCH.W[1].p06_DwnVel.xPul		:= hard.Beck[1].DIN[26];
Mc._15_WINCH.W[1].p05_UpVel.xPul		:= hard.Beck[1].DIN[27];
Mc._15_WINCH.W[1].s11_FindSeam.xPul		:= hard.Beck[1].DIN[28];
Mc._15_WINCH.W[1].s10_ControlSeam.xPul	:= hard.Beck[1].DIN[29];
Mc._15_WINCH.W[2].s10_ControlSeam.xPul	:= hard.Beck[1].DIN[30]; 
Mc._15_WINCH.W[2].s11_FindSeam.xPul		:= hard.Beck[1].DIN[31];
Mc._15_WINCH.W[2].p01_Run.xPul			:= hard.Beck[1].DIN[32]; 

(*========= MODULO 4 ===================================================*)

Mc._12_INTRO.b056_Intro_Pump.xInCons	:= hard.Beck[1].DIN[33];	
Mc._10_TK1.p150_OKprod.xPul				:= hard.Beck[1].DIN[34];
Mc._10_TK1.p151_P_Fill.xPul				:= hard.Beck[1].DIN[35];
Mc._10_TK1.P153_P_RetMc.xPul			:= hard.Beck[1].DIN[36];
Mc._10_TK1.p152_P_Drain.xPul			:= hard.Beck[1].DIN[37]; 
Mc._10_TK1.p154_P_IntroFast.xPul		:= hard.Beck[1].DIN[38];	
Mc._03_PRESS.s072_Chargr.xPul			:= hard.Beck[1].DIN[39];
Mc._03_PRESS.s073_Discharge.xPul		:= hard.Beck[1].DIN[40];
//		:= hard.Beck[1].DIN[41];
//		:= hard.Beck[1].DIN[42];
//		:= hard.Beck[1].DIN[43];
//		:= hard.Beck[1].DIN[44];
//		:= hard.Beck[1].DIN[45];
//		:= hard.Beck[1].DIN[46]; 
//		:= hard.Beck[1].DIN[47];
Mc._11_TK2.p250_OKprod.xPul				:= hard.Beck[1].DIN[48];
(*======================================================================*)
(*			DIGITAL OUTPUTS												*)
(*======================================================================*)
(*========= MODULO 5 ===================================================*)

hard.Beck[1].DOUT[1] := 			MC._00_GENERAL.p400_PMAn.xPil;
hard.Beck[1].DOUT[2] := 			MC._00_GENERAL.p401_PAuto.xPil;
hard.Beck[1].DOUT[3] := 			MC._00_GENERAL.p404_Alarm.xPil;
hard.Beck[1].DOUT[4] := 			MC._00_GENERAL.p405_Horn.xPil;
hard.Beck[1].DOUT[5] := 			MC._03_PRESS.v070_Vent.xOpen;
hard.Beck[1].DOUT[6] := 			MC._04_FILL.v002_Hot.xOpen;
hard.Beck[1].DOUT[7] := 			MC._04_FILL.v001_Cool.xOpen;
hard.Beck[1].DOUT[8] := 			MC._04_FILL.v003_Hard.xOpen;
hard.Beck[1].DOUT[9] := 			MC._05_DRAIN.v015_Grv.xOpen;
hard.Beck[1].DOUT[10] := 			MC._07_OVERFLOW.v025_Valv.xOpen;
hard.Beck[1].DOUT[11] := 			MC._02_TEMP.v061_Steam.xOpen;
hard.Beck[1].DOUT[12] := 			MC._02_TEMP.v062_Cool.xOpen;
hard.Beck[1].DOUT[13] := 			MC._02_TEMP.v063_RetCon.xOpen;
hard.Beck[1].DOUT[14] := 			MC._02_TEMP.v064_RecW.xOpen;
//hard.Beck[1].DOUT[15] := 			;
hard.Beck[1].DOUT[16] := 			MC._04_FILL.v006_InterMc.xOpen;

(*========= MODULO 6 ===================================================*)

hard.Beck[1].DOUT[17] := 			MC._09_CPUMP.b450_CircPump.xRUN;
hard.Beck[1].DOUT[18] := 			MC._15_WINCH.W[1].p00_Winch.xRUN;
//hard.Beck[1].DOUT[19] := 			MC._15_WINCH.W[1].p00_Winch.;
hard.Beck[1].DOUT[20] := 			MC._15_WINCH.W[1].p08_PilTangle.xPil;
hard.Beck[1].DOUT[21] := 			MC._15_WINCH.W[2].p00_Winch.xRUN;
//hard.Beck[1].DOUT[22] := 			MC._10_TK1.v103_IntercTK.xOpen;
hard.Beck[1].DOUT[23] := 			MC._15_WINCH.W[2].p08_PilTangle.xPil;
hard.Beck[1].DOUT[24] := 			MC._12_INTRO.b056_Intro_Pump.xRUN;
hard.Beck[1].DOUT[25] := 			MC._10_TK1.p150_OKprod.xPil;
hard.Beck[1].DOUT[26] := 			MC._10_TK1.v101_Fill.xOpen;
hard.Beck[1].DOUT[27] := 			MC._10_TK1.v102_RetMc.xOpen;
hard.Beck[1].DOUT[28] := 			MC._10_TK1.v106_Drain_grav.xOpen;
hard.Beck[1].DOUT[29] := 			MC._12_INTRO.v050_Fast.xOpen;
hard.Beck[1].DOUT[30] := 			MC._12_INTRO.v051_Slow.xOpen;
hard.Beck[1].DOUT[31] := 			MC._10_TK1.v109_Mixer.xOpen;
hard.Beck[1].DOUT[32] := 			MC._10_TK1.v107_Warm.xOpen;

(*========= MODULO 7 ===================================================*)

hard.Beck[1].DOUT[33] := 			MC._03_PRESS.v071_Load.xOpen;
hard.Beck[1].DOUT[34] := 			MC._03_PRESS.v074_Unload.xOpen;
hard.Beck[1].DOUT[35] := 			MC._07_OVERFLOW.v004_WaterInlet.xOpen;
hard.Beck[1].DOUT[36] := 			MC._08_CIRC.v044_Spray.xOpen;
hard.Beck[1].DOUT[37] := 			MC._05_DRAIN.v017_Pump.xOpen;
hard.Beck[1].DOUT[38] := 			MC._02_TEMP.v068_Purge.xOpen;
hard.Beck[1].DOUT[39] := 			MC._08_CIRC.v041_InPump.xOpen;
hard.Beck[1].DOUT[40] := 			MC._10_TK1.v103_IntercTK.xOpen;
hard.Beck[1].DOUT[41] := 			MC._11_TK2.p250_OKprod.xPil;
hard.Beck[1].DOUT[42] := 			MC._11_TK2.v201_Fill.xOpen;
hard.Beck[1].DOUT[43] := 			MC._11_TK2.v202_RetMc.xOpen;
hard.Beck[1].DOUT[44] := 			MC._11_TK2.v206_Drain_grav.xOpen;	
hard.Beck[1].DOUT[45] := 			MC._11_TK2.v203_IntercTK.xOpen;
hard.Beck[1].DOUT[46] := 			MC._11_TK2.v209_Mixer.xOpen;
hard.Beck[1].DOUT[47] := 			MC._11_TK2.v207_Warm.xOpen;;	
hard.Beck[1].DOUT[48] := 			MC._11_TK2.b204_Intro.XRun;

(*========= MODULO 8 ===================================================*)
MC._02_TEMP.s065_Reg.iAnalog		:=  hard.Beck[1].AIN[1];
//									:=  hard.Beck[1].AIN[2];		
	
(*========= MODULO 9 ===================================================*)
MC._06_LEVEL.s032_Perc.iAnalog		:=	hard.Beck[1].AIN[3];				
MC._10_TK1.s113_Level.iAnalog		:=  hard.Beck[1].AIN[4]; 	
MC._11_TK2.s213_Level.iAnalog		:=MANUAL;//:=	hard.Beck[1].AIN[5];	
Mc._03_PRESS.s075_Sensor.iAnalog	:=	hard.Beck[1].AIN[6];

(*========= MODULO 13 ==================================================*)
hard.Beck[1].AOUT[1]:=				REAL_TO_INT (Z_TEMP.rOutRegTemp);
hard.Beck[1].AOUT[2]:=				REAL_TO_INT (Z_CP.rOutAnalogVelPump);
//hard.Beck[1].AOUT[3]:=				REAL_TO_INT (_15_WINCH.W[1].rSpeedUF);
//hard.Beck[1].AOUT[4]:=				REAL_TO_INT (_15_WINCH.W[2].rSpeedUF);

END_PROGRAM

// ---- POUs/30_PLC/30_7 ActvOutputs/Modules/z_TEMP.TcPOU
PROGRAM z_TEMP

VAR
	rOutRegTemp: REAL;
END_VAR

(*-------------------------------------------------------------------------------------------------------*)
(*v061  Valvula de vapor*)
mc._02_TEMP.v061_Steam.xOpen:= F_TERMOREG.Z_xVapor OR
								F_ISOTERMA.Z_xVapor;

(*-------------------------------------------------------------------------------------------------------*)
(*v062  Valvula de enfriamiento*)
mc._02_TEMP.v062_Cool.xOpen:= F_TERMOREG.z_xEnfria OR
								F_ISOTERMA.z_xEnfria;

(*-------------------------------------------------------------------------------------------------------*)
(*v060  Apertura ValvulaModulante*)
//calentar temo
IF Mc._02_TEMP.v061_Steam.xOpen AND F_TERMOREG.xActv THEN
	Mc._02_TEMP.v060_Aper.rValue:= F_TERMOREG.z_rApertVapor;
END_IF

//calentar ISOTERMA
IF Mc._02_TEMP.v061_Steam.xOpen AND F_ISOTERMA.xActv THEN
	mc._02_TEMP.v060_Aper.rValue:= F_ISOTERMA.z_rApertVapor;
END_IF

//ENFRIAR TERMO
IF Mc._02_TEMP.v062_Cool.xOpen AND F_TERMOREG.xActv THEN
	MC._02_TEMP.v060_Aper.rValue:= F_TERMOREG.z_rApertEnfria;
END_IF

//ENFRIAR ISOTERMA
IF
	MC._02_TEMP.v062_Cool.xOpen AND F_ISOTERMA.xActv THEN
	MC._02_TEMP.v060_Aper.rValue:= F_ISOTERMA.z_rApertEnfria;
END_IF

//OUTPUT Regulacion Temperatura

rOutRegTemp:= Canvi_Escala(
				In:= mc._02_TEMP.v060_Aper.rValue, 
				In_Min:= 0, 
				In_Max:= 1, 
				Out_Min:= 0, 
				Out_Max:= 32675);
	

(*-------------------------------------------------------------------------------------------------------*)
(*v063 Retorno condensados*)
mc._02_TEMP.v063_RetCon.xOpen:= F_TERMOREG.z_xRetonoCond;

(*-------------------------------------------------------------------------------------------------------*)

END_PROGRAM

// ---- POUs/30_PLC/30_3_Config/ConfigSystem/_00_Config_PE.TcPOU
PROGRAM _00_Config_PE
VAR
	A: INT;
END_VAR

A:=A+1;

(*-------------------------------------------------------------------------------------------------------*)
(*_00_General*)
Mc._00_GENERAL.iPFTempAlta		:= WORD_TO_INT(PF[2]);		(*Temperatura para marcar temperatua alta*)

(*-------------------------------------------------------------------------------------------------------*)
(*_01_seg*)
Mc._01_SEG.iPFPresMin := 0 ;    (*FALTA DEFINIR*)
Mc._01_SEG.iPFMcMaxiTemper		:= WORD_TO_INT(PF[1]);		(*PF Maxima Temperatura Maquina*)
Mc._01_SEG.iPFTempCloseVent 	:= WORD_TO_INT(PF[3]);		(*PF Temperatura Cierra Respiradero*)
Mc._01_SEG.iPFTempBloqValv  	:= WORD_TO_INT(PF[2]);		(*PF Temperatura Bloqueo Valvulas*)
		
(*-------------------------------------------------------------------------------------------------------*)
(*_02_TEMP*)
Mc._02_TEMP.iPFDefauldGrad		:= WORD_TO_INT(PF[81]);
Mc._02_TEMP.iPFTimeOfPumpToRun	:= WORD_TO_INT(PF[82]);
Mc._02_TEMP.iPFGradIntegra		:= WORD_TO_INT(PF[83]);
Mc._02_TEMP.iPFGradForzCal		:= WORD_TO_INT(PF[84]);
Mc._02_TEMP.iPFTmpComutac		:= WORD_TO_INT(PF[85]);
Mc._02_TEMP.iPFGradComutac		:= WORD_TO_INT(PF[86]);
Mc._02_TEMP.iPFPID_P			:= WORD_TO_INT(PF[87]);
Mc._02_TEMP.iPFPID_I			:= WORD_TO_INT(PF[88]);
Mc._02_TEMP.iPFPID_D			:= WORD_TO_INT(PF[89]);
Mc._02_TEMP.iPFTempMinCool		:= WORD_TO_INT(PF[90]);


(*-------------------------------------------------------------------------------------------------------*)
(*_03_PRESS*)
Mc._03_PRESS.IPF_FS_Press 		:= WORD_TO_INT(PF[36]);
Mc._03_PRESS.iPFPresLoad 		:= WORD_TO_INT(PF[37]);
Mc._03_PRESS.IPFPresUnload 	 	:= WORD_TO_INT(PF[38]);
Mc._03_PRESS.IPFPresSeg  		:= WORD_TO_INT(PF[39]);
Mc._03_PRESS.IPFTimeOKPresSeg	:= WORD_TO_INT(PF[40]);
Mc._03_PRESS.IPFTimeDelayVent	:= WORD_TO_INT(PF[41]);

(*-------------------------------------------------------------------------------------------------------*)
(*_04_FILL*)
Mc._04_FILL.iPFFrec			  	:= WORD_TO_INT(PF[19]);		(*PF Frecuencia maxima caudalimetro*)
Mc._04_FILL.iPFFlowMax		  	:= WORD_TO_INT(PF[20]);		(*PF Caudal a la freq maxima*)
Mc._04_FILL.iPFTmClcFlow	  	:= WORD_TO_TIME(1000*PF[21]); (*PF Tiempo para el calculo de lcaudal*)
Mc._04_FILL.IPFMaxFillTime		:= PF[23];

(*-------------------------------------------------------------------------------------------------------*)
(*_05_DRAIN*)
Mc._05_DRAIN.iPFMaxTimeDrain	:= WORD_TO_INT(PF[27]) ;    //Maximo tiempo para Vaciado en seg.
Mc._05_DRAIN.iPFTimeDrenado		:= WORD_TO_INT(PF[28]) ;    //Tiempo de drenado maq. en seg.

(*-------------------------------------------------------------------------------------------------------*)
(*_06_LEVEL*)
Mc._06_LEVEL.iPFAna_min			:= WORD_TO_INT(PF[10]);		(*Ajuste minimo nivel analogico*)	
Mc._06_LEVEL.iPFAna_max			:= WORD_TO_INT(PF[11]);		(*Ajuste maximo nivel analogico*)	

Mc._06_LEVEL.iPFLvl_1			:= WORD_TO_INT(PF[14]);		(*Porcentaje del nivel para bLvl_1*)
Mc._06_LEVEL.iPFLvl_2			:= WORD_TO_INT(PF[15]);		(*Porcentaje del nivel para bLvl_2*)
Mc._06_LEVEL.iPFLvl_3			:= WORD_TO_INT(PF[16]);		(*Porcentaje del nivel para bLvl_3*)
Mc._06_LEVEL.iPFLvl_min			:= WORD_TO_INT(PF[17]);		(*Porcentaje del nivel para bLvl_min*)
Mc._06_LEVEL.iPFLvl_max			:= WORD_TO_INT(PF[18]);		(*Porcentaje del nivel para bLvl_max*)

Mc._06_LEVEL.iPFLvl_Wh			:= WORD_TO_INT(PF[12]);		(*Porcentaje del nivel bajo del lavado continuo*)
Mc._06_LEVEL.iPFLvl_Wl			:= WORD_TO_INT(PF[13]);		(*Porcentaje del nivel alto del lavado continuo*)

(*-------------------------------------------------------------------------------------------------------*)
(*_07_OVERFLOW*)
MC._07_OVERFLOW.iPFTimeFillAuxT			:= WORD_TO_INT(PF[30]);		(*Tiempo llena tank auxiliar*)	
MC._07_OVERFLOW.iPFTimeCloseAuzT		:= WORD_TO_INT(PF[31]);		(*Tiempo Fin Llenado tank auxiliar*)	
MC._07_OVERFLOW.iPFTimeDepAuxT			:= WORD_TO_INT(PF[32]);		(*Tiempo despressuriza tank aux*)	 
MC._07_OVERFLOW.iPFTimeDrainAuxT		:= WORD_TO_INT(PF[33]);		(*Tiempo Vaciado tank aux*)	
MC._07_OVERFLOW.iPFTimeCloseDrainAuxT	:= WORD_TO_INT(PF[34]);		(*Tiempo fin vaciado tank aux*)	

(*-------------------------------------------------------------------------------------------------------*)
(*_10_TK1*)
Mc._10_TK1.iPFLvlAnaMin 		:= WORD_TO_INT(PF[50]) ;
Mc._10_TK1.iPFLvlAnaMax 		:= WORD_TO_INT(PF[51]) ;
Mc._10_TK1.iPFLvlMin			:= WORD_TO_INT(PF[52]) ;
Mc._10_TK1.iPFLvlMax			:= WORD_TO_INT(PF[53]) ;
Mc._10_TK1.iPFDescSonda			:= WORD_TO_INT(PF[54]) ;
Mc._10_TK1.iPFDreno				:= WORD_TO_INT(PF[55]) ;
Mc._10_TK1.iPF1rLav				:= WORD_TO_INT(PF[56]) ;
Mc._10_TK1.iPF2nLav				:= WORD_TO_INT(PF[57]) ;
Mc._10_TK1.iPF3rLav				:= WORD_TO_INT(PF[58]) ;
Mc._10_TK1.iPFDifAlarma			:= WORD_TO_INT(PF[59]) ;
Mc._10_TK1.iPFRetarBomba		:= WORD_TO_INT(PF[60]) ;
Mc._10_TK1.iPFLowCirc			:= WORD_TO_INT(PF[61]) ;
Mc._10_TK1.iPFHighCirc			:= WORD_TO_INT(PF[62]) ;
Mc._10_TK1.iPFLvl_1				:= WORD_TO_INT(PF[63]) ;
Mc._10_TK1.iPFLvl_2				:= WORD_TO_INT(PF[64]) ;
Mc._10_TK1.iPFLvl_3				:= WORD_TO_INT(PF[65]) ;

(*-------------------------------------------------------------------------------------------------------*)
(*_11_TK2*)
Mc._11_TK2.iPFLvlAnaMin 		:= WORD_TO_INT(PF[70]) ;
Mc._11_TK2.iPFLvlAnaMax 		:= WORD_TO_INT(PF[71]) ;
Mc._11_TK2.iPFLvlMin			:= WORD_TO_INT(PF[72]) ;
Mc._11_TK2.iPFLvlMax			:= WORD_TO_INT(PF[73]) ;
Mc._11_TK2.iPFDescSonda			:= WORD_TO_INT(PF[74]) ;
Mc._11_TK2.iPFDreno				:= WORD_TO_INT(PF[75]) ;
Mc._11_TK2.iPF1rLav				:= WORD_TO_INT(PF[76]) ;
Mc._11_TK2.iPF2nLav				:= WORD_TO_INT(PF[77]) ;
Mc._11_TK2.iPF3rLav				:= WORD_TO_INT(PF[78]) ;
Mc._11_TK2.iPFDifAlarma			:= WORD_TO_INT(PF[79]) ;
Mc._11_TK2.iPFRetarBomba		:= WORD_TO_INT(PF[80]) ;
Mc._11_TK2.iPFLowCirc			:= WORD_TO_INT(PF[95]) ;
Mc._11_TK2.iPFHighCirc			:= WORD_TO_INT(PF[96]) ;
Mc._11_TK2.iPFLvl_1				:= WORD_TO_INT(PF[97]) ;
Mc._11_TK2.iPFLvl_2				:= WORD_TO_INT(PF[98]) ;
Mc._11_TK2.iPFLvl_3				:= WORD_TO_INT(PF[99]) ;

(*-------------------------------------------------------------------------------------------------------*)
(*_15_WINCH*)
Mc._15_WINCH.iPFWinchToStop		:= WORD_TO_INT(PF[31]); //Torniquete a parar en muestra (0= el primero que pase/ X= toniquete X)


Mc._15_WINCH.iPFNumSeam			:= WORD_TO_INT(PF[32]);//Numero de cuerdas
	IF Mc._15_WINCH.iPFNumSeam=0 
	THEN
	Mc._15_WINCH.iPFNumSeam:=1;
END_IF

Mc._15_WINCH.iPFNumWinch		:= WORD_TO_INT(PF[33]);//Numero de torniquetes
	IF Mc._15_WINCH.iPFNumWinch=0 
	THEN
	Mc._15_WINCH.iPFNumWinch:=1;
END_IF

Mc._15_WINCH.iPFDelayRunWinch	:= WORD_TO_INT(PF[34]);//Retraso arranque Torniquete
Mc._15_WINCH.iPFPercentWinch	:= WORD_TO_INT(PF[35]);//Porcentaje para Alarna de cuerda Parada
Mc._15_WINCH.iPFWinchMaxSpeed	:= WORD_TO_INT(PF[30]);//Velocidad Maxima torniquete
Mc._15_WINCH.iPFFactPulTor		:= WORD_TO_INT(Pf[29]);//Factor pulsadores
Mc._15_WINCH.iPFTimeMaxRope		:= WORD_TO_INT(Pf[42]);//Tiempo Maximo paso cuerda

END_PROGRAM

// ---- POUs/30_PLC/30_3_Config/ConfigSystem/_14_Config_Consum.TcPOU
PROGRAM _14_Config_Consum


(*s 500 sensor ampers para consumo*)
Mc._14_CONSUM.s500_Amperimetre.rAna_min:=0;
Mc._14_CONSUM.s500_Amperimetre.rAna_max:=37000;
Mc._14_CONSUM.s500_Amperimetre.rUf_min:=0;
Mc._14_CONSUM.s500_Amperimetre.rUf_max:=WORD_TO_REAL(PF_consum[2]);


Mc._14_CONSUM.rAmp:=Mc._14_CONSUM.s500_Amperimetre.rValue;

END_PROGRAM

// ---- POUs/30_PLC/30_3_Config/ConfigSystem/_05_Config_Drain.TcPOU
PROGRAM _05_Config_Drain
VAR
v015_Grv :fValve;
v016_Grv2 :fValve;
v017_Pump :fValve;
s018_LvlHT :dutpul;
s019_TempHT :fTemp;
v020_HT :fValve;
v021_WaterHT :fValve;
END_VAR

(*-------------------------------------------------------------------------------------------------------*)
(*-------------------------------------------------------------------------------------------------------*)

(*------------------------------------------------------------------------------------------------------*)
(*Comprobar si hay sensor de nivel del Vaciado HT *)
Mc._05_DRAIN.xLvlHT		:=Mc._05_DRAIN.s018_LvlHT.xPul;


(*Comprobar si hay PT100 del vaciado HT *)
Mc._05_DRAIN.iTempHT	:= REAL_TO_INT (Mc._05_DRAIN.s019_TempHT.rValue);



//v015_Gvr
v015_Grv(valv:=mc._05_DRAIN.v015_Grv );

//v016_Grv2
v016_Grv2 (valv:= mc._05_DRAIN.v016_Grv2);

//v017_Pump
v017_Pump(valv:=mc._05_DRAIN.v017_Pump);

//s018_LvlHT
s018_LvlHT:=mc._05_DRAIN.s018_LvlHT;
(*
//s019_TempHT 
s019_TempHT.Temp.rAna_min:=0;
s019_TempHT.Temp.rAna_max:=1500;
s019_TempHT.Temp.rUf_min:=0;
s019_TempHT.Temp.rUf_max:=150;
//s019_TempHT.Temp.
*)
//v020_HT
v020_HT(valv:=mc._05_DRAIN.v020_HT);

//v021_WaterHT
v021_WaterHT (valv:=mc._05_DRAIN.v021_WaterHT);

END_PROGRAM

// ---- POUs/40_Function_Blocks/FB/FB Duts/fValve.TcPOU
FUNCTION_BLOCK fValve

VAR_IN_OUT
	valv:dutValve;
END_VAR

VAR
	a: INT;
	tonFailFCOp: Ton;
	tonFailFCCl: Ton;
	bFailFCop:BOOL;	(*Fail FC*)
	bFailFCcl:BOOL;	(*Fail FC*)
	test: BOOL;
	tToFail: TIME := T#5S;
END_VAR

a:=a+1;

valv.xFailFC:=FALSE;
valv.xFailFCc:=FALSE;
valv.xFailFCo:=FALSE;
		
(*=========================================================================================================*)
(*Salida  BECHOFF DO*)
				
(*FC valve open*)
tonFailFCOp(IN:= (valv.xOpen)AND NOT(valv.xFailFCo) , PT:=tToFail );
valv.xFailFCo:= tonFailFCOp.Q;

(*FC valve close*)
tonFailFCCl(IN:= NOT(valv.xOpen)AND NOT(valv.xFailFCc) , PT:=tToFail  );
valv.xFailFCc:= tonFailFCCl.Q;

(*FC Valve*)		
valv.xFailFC:= valv.xFailFCo OR valv.xFailFCc;

(*=========================================================================================================*)

END_FUNCTION_BLOCK

// ---- POUs/40_Function_Blocks/FB/FB Duts/fTemp.TcPOU
FUNCTION_BLOCK fTemp
VAR_INPUT
	iAnalog:INT;
END_VAR
VAR_OUTPUT	
	rValue:REAL;
END_VAR

VAR
	A: INT;
END_VAR

(*-------------------------------------------------------------------------------------------------------*)
A:= A+1;
(*Conversion UF a temperatura ºC*)
rValue :=INT_TO_REAL(iAnalog)/10.0;

END_FUNCTION_BLOCK

// ---- POUs/30_PLC/30_3_Config/ConfigSystem/_06_Config_LEVEL.TcPOU
PROGRAM _06_Config_LEVEL
VAR
v038_FillTb :fValve;
v039_DrainTb :fValve;
	
	PresenciaNivelAnalogMc: BOOL;
	PresenciaNivelMinMc: BOOL;
	PresenciaNivelMaxMc: BOOL;
	PresenciaNivel_1_Mc: BOOL;
	PresenciaNivel_2_Mc: BOOL;
	PresenciaNivel_3_Mc: BOOL;
	NivelAltoRecircPorAnalog: BOOL;
	NivelBajoRecircPorAnalog: BOOL;
END_VAR

(*------------------------------------------------------------------------------------------------------*)
(*Configuracion nivel analogico*)

Mc._06_LEVEL.s032_Perc.rAna_max := Mc._06_LEVEL.iPFAna_max;
Mc._06_LEVEL.s032_Perc.rAna_min := Mc._06_LEVEL.iPFAna_min;

(*Comprobar si hay presencia de nivel analogico *)
PresenciaNivelAnalogMc:= TRUE;

IF PresenciaNivelAnalogMc
	THEN
		Mc._06_LEVEL.rLevel		:=Mc._06_LEVEL.s032_Perc.iAnalog;   
	ELSE
		Mc._06_LEVEL.rLevel		:= 0;		
END_IF

(*-------------------------------------------------------------------------------------------------------*)
(*Nivel Minimo*)
PresenciaNivelMinMc:= TRUE;

IF PresenciaNivelMinMc
	THEN
		Mc._06_LEVEL.xLvl_min	:= Mc._06_LEVEL.s031_Min.xPul;
	ELSIF (Mc._06_LEVEL.iPFLvl_min>0 AND NOT PresenciaNivelMinMc) THEN
		Mc._06_LEVEL.xLvl_min	:= (Mc._06_LEVEL.rLevel)>(Mc._06_LEVEL.iPFLvl_min);
	ELSE
		Mc._06_LEVEL.xLvl_min	:=FALSE;
END_IF 
(*-------------------------------------------------------------------------------------------------------*)
(*Nivel Maximo*)
PresenciaNivelMaxMc:= TRUE;
IF  PresenciaNivelMaxMc
	THEN
		Mc._06_LEVEL.xLvl_max	:= Mc._06_LEVEL.s033_max.xPul;
	ELSIF (Mc._06_LEVEL.iPFLvl_max>0 AND NOT PresenciaNivelMaxMc) THEN
		Mc._06_LEVEL.xLvl_max	:=(Mc._06_LEVEL.rLevel)>(Mc._06_LEVEL.iPFLvl_max);
	ELSE
		Mc._06_LEVEL.xLvl_max	:= FALSE;
END_IF
(*-------------------------------------------------------------------------------------------------------*)
(*Nivel 1*)
PresenciaNivel_1_Mc:= TRUE;
IF PresenciaNivel_1_Mc
	THEN
		Mc._06_LEVEL.xLvl_1	:= Mc._06_LEVEL.s036_L1.xPul;
	ELSIF (Mc._06_LEVEL.iPFLvl_1>0 AND NOT PresenciaNivel_1_Mc) THEN
		Mc._06_LEVEL.xLvl_1	:=(Mc._06_LEVEL.rLevel)>(Mc._06_LEVEL.iPFLvl_1);
	ELSE
		Mc._06_LEVEL.xLvl_1	:= FALSE;
END_IF
(*-------------------------------------------------------------------------------------------------------*)
(*Nivel 2*)
PresenciaNivel_2_Mc:=TRUE;

IF PresenciaNivel_2_Mc
	THEN
		Mc._06_LEVEL.xLvl_2	:= Mc._06_LEVEL.s035_L2.xPul;
	ELSIF (Mc._06_LEVEL.iPFLvl_2>0 AND NOT PresenciaNivel_2_Mc) THEN
		Mc._06_LEVEL.xLvl_2	:=(Mc._06_LEVEL.rLevel)>(Mc._06_LEVEL.iPFLvl_2);
	ELSE
		Mc._06_LEVEL.xLvl_2	:= FALSE;
END_IF
(*-------------------------------------------------------------------------------------------------------*)
(*Nivel 3*)
IF PresenciaNivel_3_Mc
	THEN
		Mc._06_LEVEL.xLvl_3	:= Mc._06_LEVEL.s034_L3.xPul;
	ELSIF (Mc._06_LEVEL.iPFLvl_3>0 AND NOT PresenciaNivel_2_Mc) THEN
		Mc._06_LEVEL.xLvl_3	:=(Mc._06_LEVEL.rLevel)>(Mc._06_LEVEL.iPFLvl_3);
	ELSE
		Mc._06_LEVEL.xLvl_3	:= FALSE;
END_IF
(*-------------------------------------------------------------------------------------------------------*)
(*Nivel Alto Recirculación*)
NivelAltoRecircPorAnalog:=TRUE;

IF (Mc._06_LEVEL.iPFLvl_Wh>0 AND NivelAltoRecircPorAnalog) THEN
		Mc._06_LEVEL.xLvl_Wh	:=(Mc._06_LEVEL.rLevel)>(Mc._06_LEVEL.iPFLvl_Wh);
	ELSE
		Mc._06_LEVEL.xLvl_Wh	:= Mc._06_LEVEL.xLvl_3;
END_IF
(*-------------------------------------------------------------------------------------------------------*)
(*-------------------------------------------------------------------------------------------------------*)
(*Nivel Bajo Recirculación*)
NivelBajoRecircPorAnalog:=TRUE;

IF (Mc._06_LEVEL.iPFLvl_Wl>0 AND NivelBajoRecircPorAnalog) THEN
		Mc._06_LEVEL.xLvl_Wl	:=(Mc._06_LEVEL.rLevel)>(Mc._06_LEVEL.iPFLvl_Wl);
	ELSE
		Mc._06_LEVEL.xLvl_Wl	:= Mc._06_LEVEL.xLvl_1;
END_IF

(*-------------------------------------------------------------------------------------------------------*)
(*-------------------------------------------------------------------------------------------------------*)
(*Fallo niveles*)
Mc._06_LEVEL.xFailLvl:= NOT(Mc._06_LEVEL.xLvl_min) AND
					(	Mc._06_LEVEL.xLvl_2 OR
						Mc._06_LEVEL.xLvl_3 OR
						Mc._06_LEVEL.xLvl_1 OR
						Mc._06_LEVEL.xLvl_max 
					);



(*-------------------------------------------------------------------------------------------------------*)
(*Ev Llena Indicador Nivel*)

END_PROGRAM

// ---- POUs/30_PLC/30_3_Config/ConfigSystem/_03_Config_PRESS.TcPOU
PROGRAM _03_Config_PRESS
VAR
	tOKVent: Ton;
	ExisteSensorPressMaq: BOOL;
	PressCargaDigital: BOOL;
	PressDescargaDigital: BOOL;
END_VAR


(*-------------------------------------------------------------------------------------------------------*)
(*Configuracion sensor presion*)
Mc._03_PRESS.s075_Sensor.rAna_min := 0;
Mc._03_PRESS.s075_Sensor.rAna_max := mc._03_PRESS.IPF_FS_Press ;

(*Comprobar si hay presencia de sensor presion *)
ExisteSensorPressMaq:=TRUE;

IF ExisteSensorPressMaq
	THEN
		Mc._03_PRESS.rPress		:=Mc._03_PRESS.s075_Sensor.rValue;
	ELSE
		Mc._03_PRESS.rPress		:= 0;		
END_IF

(*-------------------------------------------------------------------------------------------------------*)
(*Pression de carga*)
PressCargaDigital:=TRUE;

IF PressCargaDigital
	THEN
		Mc._03_PRESS.xPrsLoad     := Mc._03_PRESS.s072_Chargr.xPul ;
	ELSIF (Mc._03_PRESS.iPFPresLoad>0 AND NOT PressCargaDigital) THEN
		Mc._03_PRESS.xPrsLoad 	:=(Mc._03_PRESS.rPress)>(Mc._03_PRESS.iPFPresLoad );
	ELSE
		Mc._03_PRESS.xPrsLoad	:=FALSE;
END_IF


(*-------------------------------------------------------------------------------------------------------*)
(*Pression de descarga*)
PressDescargaDigital:=TRUE;
IF PressDescargaDigital
	THEN
		Mc._03_PRESS.xPrsUnload    := Mc._03_PRESS.s073_Discharge.xPul ;
	ELSIF (Mc._03_PRESS.IPFPresUnload>0 AND NOT PressDescargaDigital) THEN
		Mc._03_PRESS.xPrsUnload 	:=(Mc._03_PRESS.rPress)>(Mc._03_PRESS.IPFPresUnload );
	ELSE
		Mc._03_PRESS.xPrsUnload	:=FALSE;
END_IF

(*****************************************************************************)
//OK Respiradero por tiempo FALTA HACER POR FC o POR presion minima

tOKVent(IN:=  Mc._03_PRESS.v070_Vent.xOpen, PT:=T#5S  );
MC._03_PRESS.xOKVent := tOKVent.Q ;

END_PROGRAM

// ---- POUs/30_PLC/30_3_Config/ConfigSystem/_01_Config_SEG.TcPOU
PROGRAM _01_Config_SEG

VAR
	ExisteSenalPressMin: BOOL;
END_VAR

(*-------------------------------------------------------------------------------------------------------*)
(*Presión Mínima Máquina*)
Mc._01_SEG.xPresMin  := Mc._01_SEG.s425_PresMin.xPul ;
	

(*-------------------------------------------------------------------------------------------------------*)
(*Maxima Pression o Temperatura*)
(*Se Activa si hay entrada de maxima pression o temperatura (NC) o si la Temperatura Maq >= PF Temperatura Maxima*)
Mc._01_SEG.xMaxPresTemp  := NOT(Mc._01_SEG.s420_MaxPresTemp.xPul) OR (Mc._02_TEMP.rMacTemperature > Mc._01_SEG.iPFMcMaxiTemper);


(*-------------------------------------------------------------------------------------------------------*)
(*Temperatura Bloq. Valves*)
(*Se Activa si hay entrada de temper. bloq. valv. (NC) o si la Temperatura Maq >= PF Temperatura Maxima*)
Mc._01_SEG.xBloqValv  := NOT(Mc._01_SEG.s421_BloqValv.xPul)  OR (Mc._02_TEMP.rMacTemperature > Mc._01_SEG.iPFTempBloqValv);


(*-------------------------------------------------------------------------------------------------------*)
(*Temperatura Cierra respiradero*)
(*Se Activa si Temperatura Maq >= PF Temperatura Maxima*)
Mc._01_SEG.xTempeCloseVent	:=(Mc._02_TEMP.rMacTemperature > Mc._01_SEG.iPFTempCloseVent);      

(*-------------------------------------------------------------------------------------------------------*)
(*Maquina Cerrada*)
Mc._01_SEG.xMcClosed:=	Mc._01_SEG.s422_McClose.xPul ;      

//Alarma Maquina Abierta
Mc._01_SEG.xMcOpen:=	NOT (Mc._01_SEG.s422_McClose.xPul) AND
					(Mc._02_TEMP.rMacTemperature > MC._01_SEG.iPFTempBloqValv) ;

(*--------------------------------------------------------------------------------------*)

END_PROGRAM

// ---- POUs/30_PLC/30_3_Config/ConfigSystem/_15_Config_Winch.TcPOU
PROGRAM _15_Config_Winch
VAR
	n: INT;
	tTangle: ARRAY[1..6] OF Ton;
END_VAR

(*-------------------------------------------------------------------------------------------------------*)



(*------REPETICION POR CADA TORNIQUETE-------------------------------------------------------------------------------------------------*)
FOR n:=1 TO Mc._15_WINCH.iPFNumWinch DO
	//Enredo
	tTangle[n](	IN:= 	(*Mc.WINCH.W[n].s07_Tangle.idDI.T*)1>0 AND		//Existe la entrada de enredo
						Mc._15_WINCH.W[n].s07_Tangle.xPul , 				//Deteccion de enredo
				PT:=	T#200MS  
				);
	Mc._15_WINCH.W[n].xTangle := tTangle[n].Q;

END_FOR




(*-------REPETICION POR CADA CUERDA --------------------------------------------------------------------------------------------------*)

END_PROGRAM

// ---- POUs/30_PLC/30_3_Config/pConfig.TcPOU
PROGRAM pConfig
VAR
	a: INT;
END_VAR

(*Configuracion Entradas y Salidas*)

_14_Config_Consum();
_00_Config_General();
_00_Config_PE();
_09_Config_CPump();
_05_Config_Drain();
_04_Config_Fill();
_06_Config_LEVEL();
_07_Config_Overflow();
_03_Config_PRESS();
_01_Config_SEG();
_02_Config_TEMP();
_10_Config_TK1();
_11_Config_TK2();
_15_Config_Winch();

pIO();

UPS();

END_PROGRAM

// ---- POUs/30_PLC/30_5_Funcions/Funcions/F_AVISO.TcPOU
PROGRAM F_AVISO
VAR_INPUT
	Func:E_funcio;
	
END_VAR
VAR
	///Activa
	xActv: BOOL;
	///Fin Funcion
	xFiFunc: BOOL;
	xA_AVISO: BOOL;
	pul_FinAviso: R_trig;
	z_PilotoAlarma: BOOL;
	TON_Fi_Func: TON;
END_VAR

(*Activa funcio *)

xActv:= func.Actv_Funcio;

pul_FinAviso(CLK:=mc._00_GENERAL.p403_ContProg.xPul) ;


(*ACTIVAR SALIDAS*)
// Piloto Alarma
z_PilotoAlarma := xActv AND pul_FinAviso.Q;


(*FIN FUNCION*)
xFiFunc:= xActv AND (pul_FinAviso.Q);

(*Alarma*)
xA_AVISO:=xActv;

END_PROGRAM

// ---- POUs/30_PLC/30_5_Funcions/Funcions/F_CARGA.TcPOU
PROGRAM F_CARGA
VAR_INPUT
	Func:E_funcio;
END_VAR

VAR
	///Activa
	xActv: BOOL;
	///Fin Funcion
	xFiFunc: BOOL;
	pul_FinCarga: R_TRIG;
	xA_CARGA: BOOL;
	tempo: Ton;
	A: BOOL;
	TON_Fi_Func: TON;
	aaa: WORD;
END_VAR


xActv:= Func.Actv_Funcio;

(*Activa funcio *)
pul_FinCarga(CLK:=mc._00_GENERAL.p403_ContProg.xPul) ;

(*FIN FUNCION*)
xFiFunc:=xActv AND pul_FinCarga.Q;

(*Alarma*)
xA_CARGA:= xActv;

END_PROGRAM

// ---- POUs/30_PLC/30_5_Funcions/Funcions/F_CONTROL_PH.TcPOU
PROGRAM F_CONTROL_PH
VAR_INPUT
	Func:E_funcio;	
END_VAR
VAR
	///Activa
	xActv: BOOL;
	///Fin Funcions
	xFiFunc: BOOL;
	
	pul_FinCntlPH: R_TRIG;
	xA_CONTROL_PH: BOOL;
END_VAR


xActv:= func.Actv_Funcio;

(*Activa funcio *)

pul_FinCntlPH(CLK:=mc._00_GENERAL.p403_ContProg.xPul) ;



(*FIN FUNCION*)
xFiFunc:=xActv AND (pul_FinCntlPH.Q);

(*Alarma*)
xA_CONTROL_PH:=xActv;

END_PROGRAM

// ---- POUs/30_PLC/30_5_Funcions/Funcions/F_DESCARGA.TcPOU
PROGRAM F_DESCARGA
VAR_INPUT
	Func:E_funcio;
END_VAR
VAR
	///Activa
	xActv: BOOL;
	///Fin Funcion
	xFiFunc: BOOL;
	pul_FinDescarga: R_triG;
	xA_DESCARGA: BOOL;
END_VAR


xActv:= Func.Actv_Funcio;

(*Activa funcio *)

pul_FinDescarga(CLK:=mc._00_GENERAL.p403_ContProg.xPul) ;



(*FIN FUNCION*)
xFiFunc:=xActv AND(pul_FinDescarga.Q);

(*Alarma*)
xA_DESCARGA:=xActv;

END_PROGRAM

// ---- POUs/30_PLC/30_5_Funcions/Funcions/F_DESPRESURIZA.TcPOU
PROGRAM F_DESPRESURIZA
VAR_INPUT
	Func: E_Funcio;
END_VAR
VAR
	///Activa
	xActv: BOOL;
	///Fin Funcion
	xFinFunc: BOOL;
	
	tDespresuriza: Ton;
	xDESPRESURIZA: BOOL;
END_VAR

(*Activa funcio *)
xActv:= func.Actv_Funcio;

tDespresuriza(IN:=xActv , PT:=T#5S);



(*FIN FUNCION*)
xFinFunc					:=	xActv AND NOT (F_DESPRESURIZA.tDespresuriza.Q  OR
							Mc._03_PRESS.xOKVent
							);
xDESPRESURIZA				:=xActv;

END_PROGRAM

// ---- POUs/30_PLC/30_5_Funcions/Funcions/F_FIN_CICLO.TcPOU
PROGRAM F_FIN_CICLO
VAR_INPUT

	Func:E_funcio;
END_VAR
VAR
	///Activa
	xActv: BOOL;
	xA_FIN_CICLO: BOOL;
END_VAR

	
(* 10 Fin de ciclo*)

xActv:=func.Actv_Funcio;
ATL.PE.xEndBatch := xActv; 

(* Alarma Fin de Ciclo *)
xA_FIN_CICLO := xActv  ;

END_PROGRAM

// ---- POUs/30_PLC/30_5_Funcions/Funcions/F_INTRO_TK2.TcPOU
PROGRAM F_INTRO_TK2
VAR_INPUT
	Func:E_funcio;
END_VAR
VAR
	///Activa
	xActv: BOOL;
	///Parametros
	wP_dwTime: WORD;
	wP_dwCurve: WORD;
	wP_Wash: WORD;
	///Fin Funcion
	xFiFunc: BOOL;
	
	Intro:fB_Intro_TK;
	Wash:fBWash_TK;
	z_PumpTK: BOOL;
	z_DrainTK: BOOL;
	z_IntroSlow: BOOL;
	z_IntercepTK: BOOL;
	z_FillTK: BOOL;
	xA_TNQ_NO_OK: BOOL;
	xA_TempBloqValves: BOOL;
	xA_IntroTooSlow: BOOL;
	xA_IntroTooFast: BOOL;
	xA_BombaParadaiNTRO: BOOL;
	z_IntroFast: BOOL;
	xIntroFast: BOOL;
	tmpActivFunc: TMP_P;
	xPause:bool;
	rtCargaValores: R_trig;
	srActivIntro: SR;
	FinIntro: BOOL;
	xIntroLentaIntro: BOOL;
	xIntroRapidaIntro: BOOL;
	FinLavados: BOOL;
	xLlenaCubeta: BOOL;
	xLavadoMaquina: BOOL;
	xLavadoDreno: BOOL;
	tpFiFunc: TP;
	xIntroHT: BOOL;
	
	xIntro: BOOL;
	xDrainTk: BOOL;
	xIntercTk: BOOL;
	xPreparrIntro: BOOL;
	xFillTk: BOOL;
	xMarchaBomba: BOOL;
	tmpMarchaBomba: TMP_P;
	xPumpTk: BOOL;
	xTankNoOk: BOOL;
	xAlarmTempBloqValves: BOOL;
	rLimitInfer: REAL;
	rLimitSuper: REAL;
	TonIntroFast: TON;
	rQr: REAL;
	rQt: REAL;
	xIntroTooFast: BOOL;
	TonIntroSlow: TON;
	xIntroTooSlow: BOOL;
	CP: INT;
	xIntroRun: BOOL;
	D: TMP_P;
END_VAR

(*ACTIVAR FUNCION*)
xActv:= func.Actv_Funcio;

rtCargaValores(CLK:=xActv AND NOT xFiFunc, Q=> );

IF rtCargaValores.Q 
	THEN
	wP_dwCurve:= func.ParamFunc[1];
	wP_dwTime:= func.ParamFunc[2];
	wP_Wash:= func.ParamFunc[3];
END_IF


(********** Inicia la funcion *************)
tmpActivFunc(
	xIN:= xActv AND NOT xPause AND (F_PREP_TK2.xOK_TK OR ATL.PE.xMan) AND NOT xFiFunc,  
	xPausa:= , 
	dwSegons:= 1, 
	xQ=> , 
	dwTsegons=> , 
	rTsegons=> );

srActivIntro(SET1:=tmpActivFunc.XQ AND NOT xFiFunc, RESET:=xFiFunc OR NOT xActv, Q1=>xIntroRun );

(************** Introducion **************)
Intro(
	xActvIntro:=xIntroRun , 
	dwCurve:=wP_dwCurve , 
	dwTime:=wP_dwTime , 
	rLevel:=mc._11_TK2.rLvl , 
	xLevelMin:=mc._11_TK2.xLvl_min , 
	xIniCond:=TRUE , 
	xPause:=xPause , 
	xFiIntro=>FinIntro , 
	rQTeoric=> , 
	rQreal=> , 
	xPrepareIntro=> xPreparrIntro, 
	xDosIntro=> xIntroLentaIntro, 
	xTransferIntro=> xIntroRapidaIntro);


(************** Lavados **************)
Wash(
	xStartWash:=FinIntro , 
	xMinimLevel:=mc._11_TK2.xLvl_min , 
	dwDetectLowLevelTime:=	INT_TO_DWORD(Mc._11_TK2.iPFDescSonda) , 
	dwDrainTime:=			INT_TO_DWORD(Mc._11_TK2.iPFDreno) , 
	dw1stWashTime:=			INT_TO_DWORD(Mc._11_TK2.iPF1rLav) , 
	dw2ndWashTime:=			INT_TO_DWORD(Mc._11_TK2.iPF2nLav) , 
	dw3rdWashTime:=			INT_TO_DWORD(Mc._11_TK2.iPF3rLav) , 
	DrainType:=wP_Wash , 
	xFinWash=>FinLavados , 
	xWash=>xLlenaCubeta , 
	xToMachine=>xLavadoMaquina , 
	xToDrain=>xLavadoDreno );

	
(************** Fin Funcion **************)
xFiFunc := tpFiFunc.Q ;
tpFiFunc(IN:=FinIntro AND FinLavados , PT:=T#1S , Q=> , ET=> );

(************** Activar Salidas **************)

(* Ev Intro Rapida *)
XIntroFast := 	NOT xPause AND (xIntroRapidaIntro AND 
				(NOT MC._01_SEG.xBloqValv OR xIntroHT)) OR
				(xLavadoMaquina AND (NOT mc._01_SEG.xBloqValv OR xIntroHT));

(* Ev Intro Lenta *)
xIntro := 		NOT xPause AND (xIntroLentaIntro AND
				(NOT MC._01_SEG.xBloqValv  OR xIntroHT)) OR
				(xIntroLentaIntro AND (NOT MC._01_SEG.xBloqValv  OR xIntroHT));

(* Ev Vaciado Cubeta *)
xDrainTk := xLavadoDreno;

(* Ev Intercepta Cubeta *)
xIntercTk := xPreparrIntro OR xLavadoMaquina;	
	
(* Ev Llenado Cubeta *)
xFillTk := FinIntro AND xLlenaCubeta;

(* Bomba Intro *)
xMarchaBomba := NOT xPause AND (xPreparrIntro OR xLavadoMaquina);

tmpMarchaBomba(
	xIN:= xMarchaBomba , 
	xPausa:= , 
	dwSegons:= INT_TO_DWORD(Mc._11_TK2.iPFRetarBomba), 
	xQ=> xPumpTk, 
	dwTsegons=> , 
	rTsegons=> );

(*ACTIVAR SALIDAS*)

z_PumpTK := xPumpTk AND Mc._11_TK2.xLvl_min;

z_DrainTK := xDrainTk;

z_IntroFast := xIntroFast AND NOT Mc._01_SEG.xBloqValv AND Mc._03_PRESS.xOKVent;

z_IntroSlow := xIntro AND NOT Mc._01_SEG.xBloqValv  AND Mc._03_PRESS.xOKVent;

z_IntercepTK := xIntercTk;

z_FillTK := xFillTk;


(* Alarmas *)
// Tanq NO OK
xA_TNQ_NO_OK := xTankNoOk;

// Temperatura bloqueio de valvulas
xA_TempBloqValves := srActivIntro.Q1 AND Mc._01_SEG.xBloqValv;

// Introducion muy lenta
xA_IntroTooSlow := xIntroTooSlow;

// Introducion muy rapida
xA_IntroTooFast := xIntroTooFast;

xA_BombaParadaiNTRO:= xActv AND NOT(mC._09_CPUMP.b450_CircPump.xOK);
xTankNoOk := xActv AND NOT (F_PREP_TK2.xOK_TK OR ATL.PE.xMan);

xAlarmTempBloqValves := mc._01_SEG.xBloqValv AND NOT xIntroHT;

rLimitInfer := (1-INT_TO_REAL(Mc._11_TK2.iPFDifAlarma)/100);
rLimitSuper := (1+INT_TO_REAL(Mc._11_TK2.iPFDifAlarma)/100);

//Alarmas intro lenta o rapida
//rapida
TonIntroFast(IN:=xPreparrIntro AND (rQr < rLimitInfer*rQt) , PT:=T#20S  );
xIntroTooFast :=TonIntroFast.Q ;
//lenta
TonIntroSlow(IN:=xPreparrIntro AND (rQr > rLimitSuper*rQt) , PT:=T#20S  );
xIntroTooSlow := TonIntroSlow.Q;


//SENYALS Qt Qr per grafiques

(* Carga los valores de Intro para las graficas *)
IF 	xActv THEN 
	IF NOT(Wash.xStartWash) 
		THEN
		rQt := 100.0-Intro.rQTeoric;
		rQr := 100.0-Intro.rQreal;
		ELSE
		rQt := 100.0;
		rQr := 100.0;	
	END_IF
	ELSE
		rQt := 0;
		rQr := 0;
END_IF


Mc._11_TK2.rQt:=rQt;
Mc._11_TK2.rQr:=rQr;

END_PROGRAM

// ---- POUs/30_PLC/30_5_Funcions/Funcions/F_PREP_TK2.TcPOU
PROGRAM F_PREP_TK2
VAR_INPUT
	Func:E_funcio;
END_VAR
VAR
		///Activa
	xActv: BOOL;
	///Parametros
	wP_PrepType: WORD;
	wP_PrepPhase: WORD;
	///Fin Funcion
	xFiFunc: BOOL;
	xA_PrepareTK1: BOOL;
	z_PreAviso: BOOL;
	z_Sirena: BOOL;
	xA_PrepareTK2: BOOL;
	RESETMAN: BOOL;
	PUL: PULS_1S;
	tmpActivFunc: TMP_P;
	xResetInicio: BOOL;
	xIniciaPrep: BOOL;
	xFinPeticion: BOOL;
	xOK_TK: BOOL;
	xPedirAuto: bool;
	rsDosAuto: RS;
	xResetAuto1: BOOL;
	DosificacioAutomatica: BOOL;
	DosificacioManual: BOOL;
	xPedirMan: BOOL;
	rsDosMan: Rs;
	ResetMan1: BOOL;
	xCondOkManCub: BOOL;
	rsOKMAN: Rs;
	xOkManCub: BOOL;
	xOpCall: BOOL;
	xSirena: BOOL;
	RTPulseAuto: R_Trig;
	wRequestPhase: WORD;
	xRequestDosing: BOOL;
	xPedirDosif: BOOL;
	tOkDos: TMP_P;
	srOkDosadora: SR;
	xOkAutoCub: BOOL;
	xOK_Auto_TK: bool;
	SROkCubeta: SR;
	RESET_MAN: BOOL;
	xEnableMixer: BOOL;
	xEnableSteam: BOOL;
	xCondFiFunc: BOOL;
	TONFiFunc: TON;
END_VAR


(*ACTIVAR FUNCION*)
xActv:=func.Actv_Funcio;

wP_PrepPhase:= func.ParamFunc[1];
wP_PrepType	:= func.ParamFunc[2];


//GENERAR PULSO 1 segundo
PUL(Q=> );

//Reset inicial
tmpActivFunc(xIN:=xActv , dwSegons:=3  );
xResetInicio:=xActv AND NOT(tmpActivFunc.xQ);
//Inicia
xIniciaPrep:= tmpActivFunc.xQ;


(********Tipo Preparacion********************)
//Finalizar Petición
xFinPeticion:=	xResetInicio OR
				ATL.PE.xEndBatch OR
				ATL.PE.xStartBatch OR
				(F_INTRO_TK2.xIntroRun OR F_INTRO_TK2.srActivIntro.Q1) OR 
				xOK_TK;
		

//Auto
xPedirAuto:= (wP_PrepType=2)OR (wP_PrepType=3);
rsDosAuto(	SET:= 		xIniciaPrep	AND 
						xPedirAuto , 
			RESET1:= 	xFinPeticion OR xResetAuto1, 
			);
DosificacioAutomatica:=rsDosAuto.Q1;

//Man
xPedirMan:= (wP_PrepType=1)OR (wP_PrepType=3);
rsDosMan(	SET:= 		xIniciaPrep	AND 
						xPedirMan  , 
			RESET1:= 	xFinPeticion OR ResetMan1, 
			);
DosificacioManual:=rsDosMan.Q1;

(**************************************************************************************)	
(************************** Peticion Dosificacion Manual **************************)
(**************************************************************************************)
//Ok Dosificacion Manual
xCondOkManCub:= 	DosificacioManual AND 		//realizar Peticion manual
			MC._11_TK2.p250_OKprod.xPul AND 	//Confimacion producto
			Mc._11_TK2.xLvl_min;				//Nivel miniMO; 					 
rsOKMAN(SET:= xCondOkManCub , 
		RESET1:= NOT(Mc._11_TK2.xLvl_min) );

xOkManCub:=rsOkMan.Q1;
		
// Piloto Pre Aviso
xOpCall := (PUL.Q AND DosificacioManual AND NOT(xOkManCub)) OR xOkManCub;
// Sirena Pre Aviso para manual
xSirena := (PUL.Q AND DosificacioManual AND NOT(xOkManCub));
		

(**************************************************************************************)	
(************************** Peticion Dosificacion Automatica **************************)
(**************************************************************************************)
//Pulso inicio pedicion Auto
RTPulseAuto(CLK:= DosificacioAutomatica );

//Reset Inicial
IF xResetInicio OR RTPulseAuto.Q OR xOK_TK
	THEN
	wRequestPhase := 0;
	xRequestDosing := FALSE;
//	xOkRequest:=FALSE;
END_IF

//Pedir dosificacion
xPedirDosif:= 	DosificacioAutomatica AND NOT(ATL.PE_COM.axOkDemand[2](*XC63[1]*) OR 
				ATL.PE_COM.axOkDosage[2](*XC64[1]*));
IF xPedirDosif 
	THEN
	wRequestPhase := wP_PrepPhase;
	xRequestDosing := TRUE;
END_IF

//Confirmar Dosificacion	
tOkDos(xIN:= (ATL.PE_COM.axOkDosage[2](*XC64[1]*) ), dwSegons:=1  );
srOkDosadora(SET1:= ATL.PE_COM.axOkDosage[2](*XC64[1]*), 
			 RESET:= F_INTRO_TK2.xIntroRun OR F_INTRO_TK2.srActivIntro.Q1 OR
					xResetInicio OR 
					RTPulseAuto.Q OR
					xFinPeticion );
//OK DOS AUTO
xOkAutoCub:=srOKDosadora.Q1;					
xOK_Auto_TK:= xOkAutoCub;					

(**************************************************************************************)
(********** Ok Cubeta *************)
(**************************************************************************************)

SROkCubeta(
	SET1:= 	(wP_PrepType = 1 AND xOkManCub) OR 
			(wP_PrepType = 2 AND xOkAutoCub) OR 
			(wP_PrepType = 3 AND xOkAutoCub AND xOkManCub),
	RESET:= NOT(mc._11_TK2.xLvl_min), // OR xStartIntro,
	);

xOK_TK:=SROkCubeta.Q1 OR RESET_MAN;

IF XOK_TK 
	THEN
	xOkAutoCub:=FALSE;
	xOkManCub:=FALSE;
//	xOkRequest:=FALSE;
END_IF	





(**************************************************************************************)

(********** Agitador y Mixador *************)
xEnableMixer:=FALSE;
xEnableSteam:=FALSE;

(************** Fin Funcion **************)
xCondFiFunc := 	(rsDosAuto.Q1 AND NOT(rsDosMan.Q1) AND ATL.PE_COM.axOkDemand[2](*XC63[1]*)) OR
			(NOT(rsDosAuto.Q1) AND rsDosMan.Q1)  OR
			xOK_TK OR
			ATL.PE.xMan; 	
TONFiFunc(IN:= xCondFiFunc, PT:= T#5S );				
XFiFunc:= TONfIfUNC.Q;


IF xOK_Auto_TK OR RESETMAN THEN
	ATL.PE_COM.axOkDemand[2]:=FALSE;
	ATL.PE_COM.axOkDosage[2]:=FALSE;
	ATL.PE_COM.axDemandDos[2]:=FALSE;
	atl.PE_COM.aiNumDos[2]:=0;
END_IF


(*FINALIZAR FUNCION*)
xFiFunc:=F_PREP_TK2.xFiFunc;/////////////////////////////////////////////

	 
(*ACTIVAR SALIDAS*)
// Variables Peticion
ATL.PE_COM.axDemandDos[2] := xRequestDosing;
ATL.PE_COM.aiNumDos[2] := wRequestPhase ;
// Sirena Preaviso
z_PreAviso  :=  xOpCall;
z_Sirena 	:= 	xSirena;



(* Alarmas *)
// Pré Aviso
xA_PrepareTK2 := xSirena;

END_PROGRAM

// ---- POUs/30_PLC/30_5_Funcions/Funcions/F_LLENADO_TK2.TcPOU
PROGRAM F_LLENADO_TK2
VAR_INPUT
	Func:E_funcio;
END_VAR
VAR
		///Activa
	xActv: BOOL;
	///Parametros
	wP_RetMc: WORD;
	wP_FillLevel: WORD;
	///Fin Funcion
	xFiFunc: BOOL;
	z_05_xCleanW: BOOL;
	z_05_xMacW: BOOL;
	xA_05_TempBloqValves: BOOL;
	LlenaNivelBajo: BOOL;
	LlenaNivelMed: BOOL;
	LlenaNivelAlto: BOOL;
	LlenaNivelAnalog: BOOL;
	xLlenaAguadeRed: BOOL;
	xLlenaAguadeMaq: BOOL;
	TmpIniciaLlenado: Ton;
	SRLlenar: SR;
	xOkLlenado:BOOL;
	/// Fill Setpoint (Liters)
	wFillLiters: WORD:=0;
	RSLlenar: RS;
	TmpOK: TMP_P;
	wDelayFinFunc: WORD:=1;
	xAlarmTempBloqValves: BOOL;
	xTempBloqValves: BOOL;
	xCleanW: BOOL;
	xMacW: BOOL;
	rLitersTank: REAL:=0;
	wMc: WORD:=0;
	d: TMP_P;
	xTmpOK: BOOL;
END_VAR



(*ACTIVAR FUNCION*)
xActv:= Func.Actv_Funcio;

wP_RetMc:= Func.ParamFunc[1];
wP_FillLevel:= Func.ParamFunc[2];


IF xActv THEN
	CASE wP_FillLevel OF
		0:	
			LlenaNivelBajo := FALSE;
			LlenaNivelMed  := TRUE;
			LlenaNivelAlto := FALSE;
			LlenaNivelAnalog := FALSE;

		1:	
			LlenaNivelBajo := TRUE;
			LlenaNivelMed  := FALSE;
			LlenaNivelAlto := FALSE;
			LlenaNivelAnalog := FALSE;

		2:	
			LlenaNivelBajo := FALSE;
			LlenaNivelMed  := TRUE;
			LlenaNivelAlto := FALSE;
			LlenaNivelAnalog := FALSE;

		3:	
			LlenaNivelBajo := FALSE;
			LlenaNivelMed  := FALSE;
			LlenaNivelAlto := TRUE;
			LlenaNivelAnalog := FALSE;
		
		ELSE
			LlenaNivelBajo := FALSE;
			LlenaNivelMed  := FALSE;
			LlenaNivelAlto := FALSE;
			LlenaNivelAnalog := TRUE;	
	END_CASE
ELSE
		LlenaNivelBajo := FALSE;
		LlenaNivelMed  := FALSE;
		LlenaNivelAlto := FALSE;
		LlenaNivelAnalog := FALSE;
END_IF

(* Verfica el tipo del llenado*)
IF xActv THEN
	IF 	wP_RetMc = 0 THEN
		xLlenaAguadeRed := TRUE;
		xLlenaAguadeMaq := FALSE;
	END_IF
	IF 	wP_RetMc = 1 THEN
		xLlenaAguadeRed := FALSE;
		xLlenaAguadeMaq := TRUE;
	END_IF
ELSE
	xLlenaAguadeRed := FALSE;
	xLlenaAguadeMaq := FALSE;	
END_IF

(* Inicia el llenado*)	
TmpIniciaLlenado(IN:= xActv, PT:= T#2S, Q=> , ET=> );

SRLlenar(SET1:=TmpIniciaLlenado.Q AND NOT Mc._11_TK2.p251_P_Fill.xPul AND NOT xOkLlenado, RESET:=xTmpOk OR NOT xActv, Q1=> );

(* Finaliza el llenado por OK Llenado*)
IF NOT LlenaNivelAnalog AND LlenaNivelBajo AND (mc._11_TK2.s213_Level.rValue > INT_TO_WORD(Mc._11_TK2.iPFLvl_1)) THEN
	xOkLlenado := TRUE;
END_IF

IF NOT LlenaNivelAnalog AND LlenaNivelMed AND (mc._11_TK2.s213_Level.rValue > INT_TO_WORD (Mc._11_TK2.iPFLvl_2)) THEN
	xOkLlenado := TRUE;
END_IF

IF NOT LlenaNivelAnalog AND LlenaNivelAlto AND (mc._11_TK2.s213_Level.rValue > INT_TO_WORD (Mc._11_TK2.iPFLvl_3)) THEN
	xOkLlenado := TRUE;
END_IF

IF LlenaNivelAnalog AND(mc._11_TK2.s213_Level.rValue > wP_FillLevel) THEN
	xOkLlenado := TRUE;
END_IF

IF LlenaNivelAnalog AND wFillLiters> 0 AND (rLitersTank >= wFillLiters) THEN
	xOkLlenado := TRUE;
END_IF

IF RSLlenar.Q1 AND mc._11_TK2.s213_Level.rValue >= INT_TO_WORD (Mc._11_TK2.iPFLvlMax) THEN  
	xOkLlenado := TRUE;
END_IF

TmpOK(
	xIN:= xOkLlenado, 
	xPausa:= , 
	dwSegons:= wDelayFinFunc, 
	xQ=> xTmpOK, 
	dwTsegons=> , 
	rTsegons=> );

(* Activa salidas *)
xCleanW := SRLlenar.Q1 AND xLlenaAguadeRed AND NOT Mc._11_TK2.p251_P_Fill.xPul;
xMacW  := SRLlenar.Q1 AND xLlenaAguadeMaq AND NOT xTempBloqValves AND NOT Mc._11_TK2.p251_P_Fill.xPul;

(* Alarmas *)
xAlarmTempBloqValves := RSLlenar.Q1 AND xLlenaAguadeMaq AND xTempBloqValves;

(* Finaliza Funcion*)
xFiFunc := mc._11_TK2.xLvl_max OR xTmpOK AND NOT SRLlenar.Q1;

IF xFiFunc THEN
	xActv := FALSE;
	xOkLlenado := FALSE;
END_IF

(*ACTIVAR SALIDAS*)
// Ev. Agua Limpa
z_05_xCleanW := xCleanW AND NOT Mc._11_TK2.xLvl_max;
// Ev. Agua Maquina
z_05_xMacW := xMacW AND NOT Mc._01_SEG.xBloqValv AND NOT Mc._11_TK2.xLvl_max;



(* Alarmas *)
// Temperatura bloqueio de valvulas
xA_05_TempBloqValves := xAlarmTempBloqValves;

END_PROGRAM

// ---- POUs/30_PLC/30_5_Funcions/Funcions/F_MUESTRA.TcPOU
PROGRAM F_MUESTRA
VAR_INPUT
	Func: E_funcio;
END_VAR
VAR
	///Activa
	xActv: BOOL;
	///Fin Funcion
	xFiFunc: BOOL;
	
	pul_FinMuestra: R_trig;
	z_PilotoAlarma: BOOL;
	pul_FinAviso: R_trig;
	xA_MUESTRA: BOOL;
	rsParoTorniq: Rs;
	xParoTorniq: BOOL;
END_VAR

(*Activa funcio *)

xActv:= func.Actv_Funcio;

pul_FinMuestra(CLK:=mc._00_GENERAL.p403_ContProg.xPul) ;


(*FIN FUNCION*)
xFiFunc:=xActv AND (pul_FinMuestra.Q);


(*ACTIVAR SALIDAS*)
// Piloto Alarma
z_PilotoAlarma := xActv AND NOT  (pul_FinAviso.Q);


(*Alarma*)
xA_MUESTRA:=xActv;


//Orden Paro torniquete

rsParoTorniq(	SET:= 	 xA_MUESTRA ,  						//Activar paro con la funcion y 
						// AND Mc.WINCH.iPFWinchToStop>0 ,	//Habilitado por parametro
				RESET1:= (Mc._09_CPUMP.p451_P_Run.xPul OR 	// anular con un pulso de marcha bomba o
						NOT(Mc._09_CPUMP.p457_SelRun.xPul))	//anular deshabilitando el selector/barra
						);	
 			
xParoTorniq:=rsParoTorniq.Q1 ;

END_PROGRAM

// ---- POUs/30_PLC/30_5_Funcions/Funcions/F_PRESURIZAR.TcPOU
PROGRAM F_PRESURIZAR
VAR_INPUT
	Func:E_funcio;
END_VAR
VAR
	///Activa
	xActv: BOOL;
	///Fin Funcion
	xFinFunc: BOOL;
	
	xA_VACIADO: BOOL;
	xA_PRESURIZA: BOOL;
	z_xPresuriza: BOOL;
END_VAR

(*Activa funcio *)
xActv:= func.Actv_Funcio;

(*FIN FUNCION*)
				xFinFunc	:=	xActv AND F_DESPRESURIZA.xDESPRESURIZA;

(*ACTIVA SALIDAS*)
z_xPresuriza:= xActv  ;

END_PROGRAM

// ---- POUs/30_PLC/30_5_Funcions/Funcions/F_VACIADO_TK2.TcPOU
PROGRAM F_VACIADO_TK2
VAR_INPUT
	Func:E_funcio;
END_VAR
VAR
	///Activa
	xActv: BOOL;
	
	z_xValVaciado: BOOL;
	z_BombaVaciado: BOOL;
	tBombaTk: Ton;
	xFiFunc: BOOL;
	xDrainTk: BOOL;
	srActivaVaciado: SR;
	xVaciar: bool;
	tVacia: TMP_P;
	tMarchaBomba: TON;
	tFinF: TP;
	D: TON;
END_VAR


(*ACTIVA FUNCIÓN*)
xActv:=func.Actv_Funcio;


srActivaVaciado(SET1:=xActv AND NOT xFiFunc, RESET:= xFiFunc OR NOT xActv ,Q1=> );

xVaciar := srActivaVaciado.Q1 AND NOT tVacia.XQ;

tVacia(
	xIN:= srActivaVaciado.Q1 AND NOT MC._11_TK2.xLvl_min, 
	xPausa:= , 
	dwSegons:= INT_TO_WORD(Mc._11_TK2.iPFDreno) , 
	xQ=> , 
	dwTsegons=> , 
	rTsegons=> );

tMarchaBomba(IN:= xVaciar, PT:= T#2S, Q=> , ET=> );	

(* Ev Vaciado Cubeta *)
xDrainTk := xVaciar;

tFinF(IN:= tVacia.XQ, PT:=T#1S , Q=>xFiFunc , ET=> );

IF xFiFunc THEN
	xActv := FALSE;
END_IF


(* FINALIZAR LA FUNCION *)
xFiFunc:= F_VACIADO_TK2.xFiFunc;

(*ACTIVAR SALIDA*)

z_xValVaciado:=xDrainTk;

tBombaTk(IN:= z_xValVaciado, PT:=INT_TO_TIME(Mc._11_TK2.iPFRetarBomba*1000) );

z_BombaVaciado:=tBombaTk.Q;

END_PROGRAM

// ---- POUs/30_PLC/30_5_Funcions/Funcions/F_VELOCIDADES.TcPOU
PROGRAM F_VELOCIDADES
VAR_INPUT
	Func:E_Funcio;
END_VAR
VAR
	///Activa
	xActv: BOOL;
	///Parametros
	wP_SP_SpeedPumpC: WORD;
	wP_SP_Speed: WORD;
	wP_SP_T_Pass: WORD;
	///Fin Funcion
	xFinFunc: BOOL;
	tFinFuncion: Ton;
	a: INT;
	rOutAnalogSpeedPumpC: REAL;
END_VAR


a:=a+1;

(*Activa funcio *)
xActv:= func.Actv_Funcio;

wP_SP_SpeedPumpC:= func.ParamFunc[1];
wP_SP_Speed:= func.ParamFunc[2];
wP_SP_T_Pass:= func.ParamFunc[3];

(*
IF xActv
	THEN
	(*Torniquets*)
	IF wP_SP_Speed>0 THEN
		Mc.WINCH.iSP_Speed:=WORD_TO_INT(wP_SP_Speed);
	END_IF

	IF wP_SP_T_Pass>0 THEN
		Mc.WINCH.iSP_T_Pass:=WORD_TO_INT(wP_SP_T_Pass);
	END_IF
	*)

(*Bomba*)
IF wP_SP_SpeedPumpC >0 THEN
		mc._08_CIRC.rSP_SpeedPumpC:=  Canvi_Escala(
													In:= wP_SP_SpeedPumpC, 
													In_Min:= Mc._09_CPUMP.iPF_AnaMin_UF, 
													In_Max:= Mc._09_CPUMP.iPF_AnaMax_UF, 
													Out_Min:= 0, 
													Out_Max:= 100);
END_IF
	
		
(*Fin funcio *)
tFinFuncion(IN:=xActv , PT:=T#5S);
xFinFunc:= tFinFuncion.Q;

END_PROGRAM

// ---- POUs/30_PLC/30_5_Funcions/Funcions/_00_GENERALES.TcPOU
PROGRAM _00_GENERALES
VAR
	Pulso_1s: fbpulse1s;
	
END_VAR

//GENERA PULSOS Y FLANCOS CADA SEGUNDO

Pulso_1s ();

END_PROGRAM

// ---- POUs/30_PLC/30_5_Funcions/Funcions/_00_GESTION_PUL.TcPOU
PROGRAM _00_GESTION_PUL
VAR
	pPulseFillTK1: R_trig;
	RS_ActiveFillTK1: RS;
	xOKFillTK1: BOOL;
	z_FillTK1Manual: BOOL;
	pPulseDrainTK1: R_TRIG;
	xOKDrainTK1: BOOL;
	z_DrainTK1Manual: BOOL;
	RS_ActiveDrainTK1: RS;
	pPulseRut1: R_trig;
	pPulseRetourn: R_trig;
	RsRetounTK1: RS;
	xOkRetournTK1: BOOL;
	z_RetMcTk1Manual: BOOL;
	pPulseSlowIntro: R_trig;
	RsSlowIntroTK1: rs;
	xOkSlowIntroTK1: BOOL;
	z_IntroSlowManual: BOOL;
	xA_RutinaActv: BOOL;
	pPulseFastIntro: R_trig;
	RsFastIntroTK1: Rs;
	z_IntroFastManual: BOOL;
	xOkFastIntroTK1: BOOL;
	tDrenado: Ton;
	pPulseLavTub: R_trig;
	RsLavTuberias: Rs;
	xLavTuberias: BOOL;
	z_LavTuberias: BOOL;
	tDrenadoColores: Ton;
	pPulseTransMaq: R_trig;
	RsTransMaq: Rs;
	xTransMaq: BOOL;
	z_TransMaq: BOOL;
	pPulseTransTk1: R_trig;
	xTransTK1: BOOL;
	z_TransTK1: BOOL;
	RsTransTK1: Rs;
	tDrenadoVac: Ton;
	tDrenadoIntroR: Ton;
	tDrenadoIntroL: Ton;
	tDrenadoColLTs: Ton;
	tDrenadoColTMc: Ton;
	tDrenadoColTK1: Ton;
	pPulseLlenadoTKC: R_trig;
	RsLlenTKC: Rs;
	xLlenaTKC: BOOL;
	z_LlenaTKC: BOOL;
	pPulseVaciaTkc: R_trig;
	tDrenadoColVac: Ton;
	xVaciaTKC: BOOL;
	RsVaciaTKC: Rs;
	z_VaciaTKC: BOOL;
	pPulseFillTK2: R_trig;
	RS_ActiveFillTK2: RS;
	xOKFillTK2: BOOL;
	z_FillTK2Manual: BOOL;
	pPulseDrainTK2: R_TRIG;
	tDrenadoVacTK2: TON;
	xOKDrainTK2: BOOL;
	RS_ActiveDrainTK2: RS;
	z_DrainTK2Manual: BOOL;
	pPulseRetournTK2: R_TRIG;
	RsRetounTK2: RS;
	xOkRetournTK2: BOOL;
	tDrenadoTK2: TON;
	z_RetMcTk2Manual: BOOL;
	tDrenadoIntroRTK2: TON;
	xOkFastIntroTK2: BOOL;
	RsFastIntroTK2: RS;
	pPulseFastIntroTK2: R_TRIG;
	z_IntroFastManualTK2: BOOL;
	pPulsesLOWIntroTK2: R_TRIG;
	tDrenadoIntroLTK2: TON;
	xOkSLOWIntroTK2: BOOL;
	z_IntroSlowManualTK2: BOOL;
	pPulseEvMixer: R_trig;
	RsMixerTK1: RS;
	xOkMixerTK1: BOOL;
	z_MixerTk1Manual: BOOL;
	RsMixerTK2: RS;
	pPulseEvMixerTK2: R_TRIG;
	xOkMixerTK2: BOOL;
	z_MixerTk2Manual: BOOL;
	pPulsoVaporTK1: R_TRIG;
	RsVaporTK1: RS;
	xOkVaporTK1: BOOL;
	z_VaporTk1Manual: BOOL;
END_VAR

//++++++++++++++++++++++++++++++++++++++++++++++++++++++++++++++++++++++++++++
//  			TK1 TK1 TK1
//++++++++++++++++++++++++++++++++++++++++++++++++++++++++++++++++++++++++++++
(*
//Calcular tiempo drenado
tDrenado(IN:=NOT(Mc.TK1.xLvl_min) , PT:= INT_TO_TIME(Mc.TK1.iPFDreno)*1000  );



// Rutina LLenado TK1 Manual

pPulseFillTK1(CLK:= MC.TK1.p151_P_Fill.bPul , Q=> );				//Pulso llenado cubeta manual

RS_ActiveFillTK1(SET:= pPulseFillTK1.Q AND NOT xOKFillTK1, //Activa por pulsador
				RESET1:= (pPulseFillTK1.Q AND xOKFillTK1)  //Resetea por pulsador
				OR MC.TK1.xLvl_3 , 						   //Resetea por llegar a nivel 1
				Q1=> xOKFillTK1 );

z_FillTK1Manual:= xOKFillTK1;


// Rutina Vaciado TK1 Manual

pPulseDrainTK1(CLK:= MC.TK1.p152_P_Drain.bPul , Q=> );				//Pulso Vaciado cubeta manual
//Calcular tiempo drenado
tDrenadoVac(IN:=xOKDrainTK1 AND NOT(Mc.TK1.xLvl_min) , PT:= INT_TO_TIME(Mc.TK1.iPFDreno)*1000  );

RS_ActiveDrainTK1(	SET:= 	pPulseDrainTK1.Q AND 
							NOT xOKDrainTK1, //Activa por pulsador
					RESET1:= (pPulseDrainTK1.Q AND xOKDrainTK1)  OR //Resetea por pulsador
							tDrenadoVac.Q , 		//Resetea si no tiene nivel mínimo
					Q1=> xOKDrainTK1 );

z_DrainTK1Manual:= xOKDrainTK1;


// Activa Retorno TK1 Manual

pPulseRetourn(CLK:=MC.TK1.P153_P_RetMc.bPul, Q=> ); //Pulso para activación Retorno TK1 Manual

RsRetounTK1(	SET:= pPulseRetourn.Q AND 
						NOT xOkRetournTK1,          //Start Retorno TK1 por pulsador
				RESET1:= (pPulseRetourn.Q AND
						 xOkRetournTK1)OR			//Stop retorno TK1 por pulsador
						MC.SEG.xBloqValv OR
						mc.TK1.xLvl_max	,			//Stop retorno TK1 por nivel minimo
				Q1=> xOkRetournTK1 );

z_RetMcTk1Manual:= xOkRetournTK1;

// Activa Intro Rapida TK1 Manual

pPulseFastIntro(CLK:=MC.TK1.p154_P_IntroFast.bPul  ); //Pulso para activación Intro Lenta Manual
//Calcular tiempo drenado
tDrenadoIntroR(IN:=xOkFastIntroTK1 AND NOT(Mc.TK1.xLvl_min) , PT:= INT_TO_TIME(Mc.TK1.iPFDescSonda)*1000  );

RsFastIntroTK1(	SET:= pPulseFastIntro.Q AND 
						NOT xOkFastIntroTK1 AND //Start Slow Intro TK1 por pulsador
						mc.TK1.xLvl_min,        //Asegura nivel mínimo TK1
				RESET1:= (pPulseFastIntro.Q AND
						 xOkFastIntroTK1) OR 			//Stop retorno TK1 por Temp.Bloq.Valv
						 tDrenadoIntroR.Q	,	
				Q1=> xOkFastIntroTK1);

z_IntroFastManual:= xOkFastIntroTK1;


// Activa Intro lenta TK1 Manual

pPulsesLOWIntro(CLK:=MC.TK1.p156_P_IntroSlow.bPul  ); //Pulso para activación Intro Lenta Manual
//Calcular tiempo drenado
tDrenadoIntroL(IN:=xOkSLOWIntroTK1 AND NOT(Mc.TK1.xLvl_min) , PT:= INT_TO_TIME(Mc.TK1.iPFDreno)*1000  );
RsSlowIntroTK1(	SET:= pPulseSlowIntro.Q AND 
						NOT xOkSlowIntroTK1 AND	//Start Slow Intro TK1 por pulsador
						MC.TK1.xLvl_min,        //Asegura nivel mínimo TK1
				RESET1:= (pPulseSlowIntro.Q AND
						 xOkSlowIntroTK1) OR 			//Stop retorno TK1 por Temp.Bloq.Valv
						 tDrenadoIntroL.Q	,	
				Q1=> xOkSlowIntroTK1);

z_IntroSlowManual:= xOkSlowIntroTK1;

// Activa Mezcla TK1

pPulseEvMixer(CLK:=MC.TK1.p158_P_Mixer.bPul, Q=> ); //Pulso para activación EV Mixer TK1 Manual

RsMixerTK1(	SET:= pPulseEvMixer.Q AND NOT 			//Start Ev Mixer TK1 por pulsador
					xOkMixerTK1 AND NOT
					xOkMixerTK2,        			//No permite Start si mixer TK2 Activo
				RESET1:=(pPulseEvMixer.Q AND
						xOkMixerTK1)OR				//Stop Ev Mixer TK1 por pulsador
						mc.TK1.xLvl_max OR NOT		//Stop Ev Mixer TK1 por nivel máximo
						mc.TK1.xLvl_min OR			//Stop Ev Mixer TK1 por nivel mínimo
						F_INTRO_TK1.xActv OR		//Stop Ev Mixer TK1 si Funcion Intro TK1 Activa
						F_INTRO_TK2.xActv	,		//Stop Ev Mixer TK1 si Funcion Intro TK2 Activa
				Q1=> xOkMixerTK1 );

z_MixerTk1Manual:=  xOkMixerTK1;

// Activa Mezcla TK1

pPulsoVaporTK1(CLK:=MC.TK1.p155_P_Warm.bPul, Q=> ); //Pulso para activación EV Calentar TK1 Manual

RsVaporTK1(	SET:= 	pPulsoVaporTK1.Q AND NOT 		//Start Calentar TK1 MANUAL
					xOkVaporTK1, 	       			//No permite Start si mixer TK2 Activo
				RESET1:=(pPulsoVaporTK1.Q AND
						xOkVaporTK1)OR	NOT			//Stop Ev Vapor TK1 por pulsador
						Mc.TK1.xLvl_2,			//Stop Ev Vapor TK1 por nivel mínimo
				Q1=> xOkVaporTK1 );

z_VaporTk1Manual:=  xOkVaporTK1;

*)

//++++++++++++++++++++++++++++++++++++++++++++++++++++++++++++++++++++++++++++
//  			TK2 TK2 TK2
//++++++++++++++++++++++++++++++++++++++++++++++++++++++++++++++++++++++++++++

//Calcular tiempo drenado
tDrenadoTK2(IN:=NOT(Mc._11_TK2.xLvl_min) , PT:= INT_TO_TIME(Mc._11_TK2.iPFDreno)*1000  );



// Rutina LLenado TK2 Manual

pPulseFillTK2(CLK:= MC._11_TK2.p251_P_Fill.xPul , Q=> );		//Pulso llenado cubeta manual

RS_ActiveFillTK2(SET:= pPulseFillTK2.Q AND NOT xOKFillTK2, //Activa por pulsador
				RESET1:= (pPulseFillTK2.Q AND xOKFillTK2)  //Resetea por pulsador
				OR MC._11_TK2.xLvl_3 , 						   //Resetea por llegar a nivel 1
				Q1=> xOKFillTK2 );

z_FillTK2Manual:= xOKFillTK2;


// Rutina Vaciado TK2 Manual

pPulseDrainTK2(CLK:= MC._11_TK2.p252_P_Drain.xPul , Q=> );				//Pulso Vaciado cubeta manual
//Calcular tiempo drenado
tDrenadoVacTK2(IN:=xOKDrainTK2 AND NOT(Mc._11_TK2.xLvl_min) , PT:= INT_TO_TIME(Mc._11_TK2.iPFDreno)*1000  );

RS_ActiveDrainTK2(	SET:= 	 pPulseDrainTK2.Q AND 
							 NOT xOKDrainTK2, 						//Activa por pulsador
					RESET1:= (pPulseDrainTK2.Q AND xOKDrainTK2)  OR //Resetea por pulsador
							 tDrenadoVacTK2.Q , 					//Resetea si no tiene nivel mínimo
					Q1=> xOKDrainTK2 );

z_DrainTK2Manual:= xOKDrainTK2;


// Activa Retorno TK2 Manual

pPulseRetournTK2(CLK:=MC._11_TK2.P253_P_RetMc.xPul, Q=> ); //Pulso para activación Retorno TK1 Manual

RsRetounTK2(	SET:= pPulseRetournTK2.Q AND 
						NOT xOkRetournTK2,          //Start Retorno TK1 por pulsador
				RESET1:= (pPulseRetournTK2.Q AND
						 xOkRetournTK2)OR			//Stop retorno TK1 por pulsador
						MC._01_SEG.xBloqValv OR
						mc._11_TK2.xLvl_max	,			//Stop retorno TK1 por nivel minimo
				Q1=> xOkRetournTK2 );

z_RetMcTk2Manual:= xOkRetournTK2;

// Activa Intro Rapida TK2 Manual

pPulseFastIntroTK2(CLK:=MC._11_TK2.p254_P_IntroFast.xPul  ); //Pulso para activación Intro Lenta Manual
//Calcular tiempo drenado
tDrenadoIntroRTK2(IN:=xOkFastIntroTK2 AND NOT(Mc._11_TK2.xLvl_min) , PT:= INT_TO_TIME(Mc._11_TK2.iPFDescSonda)*1000  );

RsFastIntroTK2(	SET:= 	pPulseFastIntroTK2.Q AND 
						NOT xOkFastIntroTK2 AND 
						mc._11_TK2.xLvl_min,        	//Start Slow Intro TK1 por pulsador
				RESET1:= (pPulseFastIntroTK2.Q AND
						 xOkFastIntroTK2) OR 			//Stop retorno TK1 por Temp.Bloq.Valv
						 tDrenadoIntroRTK2.Q 	,	
				Q1=> 	 xOkFastIntroTK2);

z_IntroFastManualTK2:= xOkFastIntroTK2;


// Activa Intro lenta TK2 Manual

pPulsesLOWIntroTK2(CLK:=MC._11_TK2.p256_P_IntroSlow.xPul  ); //Pulso para activación Intro Lenta Manual
//Calcular tiempo drenado
tDrenadoIntroLTK2(IN:=xOkSLOWIntroTK2 AND NOT(Mc._11_TK2.xLvl_min) , PT:= INT_TO_TIME(Mc._11_TK2.iPFDreno)*1000  );
RsSlowIntroTK1(	SET:= pPulseSlowIntroTK2.Q AND 
						NOT xOkSlowIntroTK2,        //Start Slow Intro TK1 por pulsador
				RESET1:= (pPulseSlowIntroTK2.Q AND
						 xOkSlowIntroTK2) OR 			//Stop retorno TK1 por Temp.Bloq.Valv
						 tDrenadoIntroLTK2.Q	,	
				Q1=> xOkSlowIntroTK2);

z_IntroSlowManualTK2:= xOkSlowIntroTK2;

// Activa Mezcla TK2

pPulseEvMixerTK2(CLK:=MC._11_TK2.p258_P_Mixer.xPul, Q=> ); //Pulso para activación EV Mixer TK2 Manual

RsMixerTK2(	SET:= pPulseEvMixerTK2.Q AND NOT     	//Start Ev Mixer TK2 por pulsador
				 		xOkMixerTK2 AND NOT
						xOkMixerTK1,             	//No permite Start si mixer TK1 Activo
				RESET1:=(pPulseEvMixerTK2.Q AND
						xOkMixerTK2)OR				//Stop Ev Mixer TK2 por pulsador
						mc._11_TK2.xLvl_max OR NOT		//Stop Ev Mixer TK2 por nivel máximo
						mc._11_TK2.xLvl_min OR			//Stop Ev Mixer TK2 por nivel mínimo
						//F_INTRO_TK1.xActv OR		//Stop Ev Mixer TK2 si Funcion Intro TK1 Activa
						F_INTRO_TK2.xActv	,		//Stop Ev Mixer TK2 si Funcion Intro TK2 Activa
				Q1=> xOkMixerTK2 );

z_MixerTk2Manual:= xOkMixerTK2;

//Rutina activa
xA_RutinaActv:=  xOKFillTK1 OR
				xOKDrainTK1 OR
				xOkRetournTK1 OR
				xOkSlowIntroTK1	OR
				xOkFastIntroTK1 OR
				xOKFillTK2 OR
				xOKDrainTK2 OR
				xOkRetournTK2 OR
				xOkSlowIntroTK2 OR
				xOKFastIntroTK2;

(*
//++++++++++++++++++++++++++++++++++++++++++++++++++++++++++++++++++++++++++++
//  			TKC TKC TKC
//++++++++++++++++++++++++++++++++++++++++++++++++++++++++++++++++++++++++++++

//Drenado cocina colores


//Calcular tiempo drenado
tDrenadoColores(IN:=NOT(Mc.TKC.xLvl_min) , PT:= INT_TO_TIME(Mc.TKC.iPFDreno)*1000  );

//------------------------------------------------------------

// Lavado tuberias
pPulseLavTub(CLK:=MC.TKC.p351_Pul_LavTub.bPul  ); //Pulso para activación Intro Lenta Manual
//Calcular tiempo drenado
tDrenadoColLTs(IN:=xLavTuberias AND NOT(Mc.TKC.xLvl_min) , PT:= INT_TO_TIME(Mc.TKC.iPFDreno)*1000  );

RsLavTuberias(	SET:= pPulseLavTub.Q AND 
						NOT xLavTuberias,        //Start Slow Intro TK1 por pulsador
				RESET1:= (pPulseLavTub.Q AND
						 xLavTuberias) OR 			//Stop retorno TK1 por Temp.Bloq.Valv
						 tDrenadoColLTs.Q	,	
				Q1=> xLavTuberias);

//Salidas
z_LavTuberias:= xLavTuberias;
Mc.TKC.p351_Pul_LavTub.bPilot:= xLavTuberias ;
//------------------------------------------------------------

// Transferencia maquina
pPulseTransMaq(CLK:=MC.TKC.p352_Pul_TransMaq.bPul  ); //Pulso para activación Intro Lenta Manual
//Calcular tiempo drenado
tDrenadoColTMc(IN:=xTransMaq AND NOT(Mc.TKC.xLvl_min) , PT:= INT_TO_TIME(Mc.TKC.iPFDreno)*1000  );

RsTransMaq(		SET:= 	pPulseTransMaq.Q AND 
						NOT xTransMaq,        //Start Slow Intro TK1 por pulsador
				RESET1:= (pPulseTransMaq.Q AND
						 xTransMaq) OR 			//Stop retorno TK1 por Temp.Bloq.Valv
						 tDrenadoColTMc.Q	,	
				Q1=> 	xTransMaq);

//Salidas
z_TransMaq:= xTransMaq;
Mc.TKC.p352_Pul_TransMaq.bPilot:= xTransMaq ;
//------------------------------------------------------------

// Transferencia tanque
pPulseTransTk1(CLK:=MC.TKC.p353_Pul_TransTanque.bPul  ); //Pulso para activación Intro Lenta Manual
//Calcular tiempo drenado
tDrenadoColTK1(IN:=xTransTK1 AND NOT(Mc.TKC.xLvl_min) , PT:= INT_TO_TIME(Mc.TKC.iPFDreno)*1000  );

RsTransTK1(		SET:= 	pPulseTransTk1.Q AND 
						NOT xTransTK1,        //Start Slow Intro TK1 por pulsador
				RESET1:= (pPulseTransTk1.Q AND
						 xTransTK1) OR 			//Stop retorno TK1 por Temp.Bloq.Valv
						 tDrenadoColTK1.Q	,	
				Q1=> 	xTransTK1);

//Salidas
z_TransTK1:= xTransTK1;
Mc.TKC.p353_Pul_TransTanque.bPilot:= xTransTK1 ;
//------------------------------------------------------------

// Llenado tanque Color
pPulseLlenadoTKC(CLK:=MC.TKC.p354_Pul_llenado.bPul  ); //Pulso para activación 

RsLlenTKC(		SET:= 	pPulseLlenadoTKC.Q AND 
						NOT xLlenaTKC,        //Start Slow Intro TK1 por pulsador
				RESET1:= (pPulseLlenadoTKC.Q AND
						 xLlenaTKC) OR 			//Stop retorno TK1 por Temp.Bloq.Valv
						 Mc.TKC.xLvl_max	,	
				Q1=> 	xLlenaTKC);

//Salidas
z_LlenaTKC:= xLlenaTKC;





//------------------------------------------------------------

// Vaciado tanque
pPulseVaciaTkc(CLK:=MC.TKC.p355_Pul_Vaciado.bPul  ); //Pulso para activación 
//Calcular tiempo drenado
tDrenadoColVac(IN:=xVaciaTKC AND NOT(Mc.TKC.xLvl_min) , PT:= INT_TO_TIME(Mc.TKC.iPFDreno)*1000  );

RsVaciaTKC(		SET:= 	pPulseVaciaTkc.Q AND 
						NOT xVaciaTKC,        //Start Slow Intro TK1 por pulsador
				RESET1:= (pPulseVaciaTkc.Q AND
						 xVaciaTKC) OR 			//Stop retorno TK1 por Temp.Bloq.Valv
						 tDrenadoColVac.Q	,	
				Q1=> 	xVaciaTKC);

//Salidas
z_VaciaTKC:= xVaciaTKC;
 //------------------------------------------------------------*)

END_PROGRAM

// ---- POUs/30_PLC/30_5_Funcions/Funcions/_00_VENT.TcPOU
PROGRAM _00_VENT
VAR
	xVentFunc: BOOL;
	xPresuriza: BOOL;
	Z_xDescarga: BOOL;
	tPresuriza: Ton;
	tDelayDescarga: TIME := TIME#2s0ms;
	tDelayRespira: TIME := TIME#2s0ms;
	tRespira: Ton;
	z_xRespiradero: BOOL;
	z_xCargaPres: BOOL;
	xDespresuriz: BOOL;
	xDescargaHighPress: BOOL;
	xDescargaPorResp: BOOL;
END_VAR

//Activar Respiradero por Funcion
xVentFunc:= F_LLENADO.z_xActvVent OR
			F_LAVADO_CONT.z_xActvVent OR	
			F_VACIADO.z_xActvVent      
			;								

